# B&R Automation Studio project NAELD004C00R10L518F00 (part 25)

#### Local.var
```iecst
(*2023-02-13*)
(**)
(*Local Action, State & Status*)
VAR
	eAct : eMagRcpAction := MagRcpActIdle;
	eStat : eMagRcpAction := MagRcpActIdle;
	eStatus : eFBStatus := Idle;
	udiStatus : UDINT := 0;
	sStatTxt : STRING[200] := '';
	a_sStatText : ARRAY[0..50] OF STRING[200] := ['Idling','Creating Directory','Adding and Editing Files','Deleting Files','Get Info','Get List','Filtering Files','Reading Current Recipe','Loading Current Recipe','Writing Current Recipe Parameter','Saving List',40('')];
END_VAR
(**)
(*Local Alarm*)
VAR
	tyAlmData : tyAlmDat;
	a_tyAlmText : ARRAY[10000..10099] OF tyAlmTxt := [(sAlmText:='Create User Directory Error',sRcyText:='Unable To Create User Directory. Please Contact Nutek For A Possible Solution'),(sAlmText:='Create Magazine Recipe Directory Error',sRcyText:='Unable To Create Magazine Recipe Directory. Please Contact Nutek For A Possible Solution'),(sAlmText:='File Open Error While Adding & Editing',sRcyText:='An Error Was Encountered While Trying To Open File. Please Contact Nutek For A Possible Solution.'),(sAlmText:='File Create Error While Adding & Editing',sRcyText:='An Error Was Encountered While Trying To Create File. Please Contact Nutek For A Possible Solution.'),(sAlmText:='File Write Error While Adding & Editing',sRcyText:='An Error Was Encountered While Trying To Write File. Please Contact Nutek For A Possible Solution.'),(sAlmText:='File Close Error While Adding & Editing',sRcyText:='An Error Was Encountered While Trying To Close File. Please Contact Nutek For A Possible Solution.'),(sAlmText:='File Open Error While Deleting',sRcyText:='An Error Was Encountered While Trying To Open File. Please Contact Nutek For A Possible Solution.'),(sAlmText:='File Create Error While Deleting',sRcyText:='An Error Was Encountered While Trying To Create File. Please Contact Nutek For A Possible Solution.'),(sAlmText:='File Write Error While Deleting',sRcyText:='An Error Was Encountered While Trying To Write File. Please Contact Nutek For A Possible Solution.'),(sAlmText:='File Close Error While Deleting',sRcyText:='An Error Was Encountered While Trying To Close File. Please Contact Nutek For A Possible Solution.'),(sAlmText:='File Open Error While Getting List',sRcyText:='An Error Was Encountered While Trying To Open File. Please Contact Nutek For A Possible Solution.'),(sAlmText:='File Read Error While Getting List',sRcyText:='An Error Was Encountered While Trying To Read File. Please Contact Nutek For A Possible Solution.'),(sAlmText:='File Close Error While Getting List',sRcyText:='An Error Was Encountered While Trying To Close File. Please Contact Nutek For A Possible Solution.'),(sAlmText:='Directory Does Not Exist While Adding & Editing',sRcyText:='The Directory Does Not Exist.Please Contact Nutek For A Possible Solution.'),(sAlmText:='Directory Does Not Exist While Deleting',sRcyText:='The Directory Does Not Exist.Please Contact Nutek For A Possible Solution.'),(sAlmText:='File Open Error While Loading Current Recipe',sRcyText:='An Error Was Encountered While Trying To Open File. Please Contact Nutek For A Possible Solution.'),(sAlmText:='File Create Error While Loading Current Recipe',sRcyText:='An Error Was Encountered While Trying To Create File. Please Contact Nutek For A Possible Solution.'),(sAlmText:='File Write Error While Loading Current Recipe',sRcyText:='An Error Was Encountered While Trying To Write File. Please Contact Nutek For A Possible Solution.'),(sAlmText:='File Close Error While Loading Current Recipe',sRcyText:='An Error Was Encountered While Trying To Close File. Please Contact Nutek For A Possible Solution.'),(sAlmText:='Directory Does Not Exist While Loading Current Recipe',sRcyText:='The Directory Does Not Exist.Please Contact Nutek For A Possible Solution.'),(sAlmText:='File Open Error While Reading Current Recipe',sRcyText:='An Error Was Encountered While Trying To Open File. Please Contact Nutek For A Possible Solution.'),(sAlmText:='File Read Error While Reading Current Recipe',sRcyText:='An Error Was Encountered While Trying To Read File. Please Contact Nutek For A Possible Solution.'),(sAlmText:='File Close Error While Reading Current Recipe',sRcyText:='An Error Was Encountered While Trying To Close File. Please Contact Nutek For A Possible Solution.'),(sAlmText:='File Open Error While Writing Current Recipe Parameter',sRcyText:='An Error Was Encountered While Trying To Open File. Please Contact Nutek For A Possible Solution.'),(sAlmText:='File Create Error While Writing Current Recipe Parameter',sRcyText:='An Error Was Encountered While Trying To Create File. Please Contact Nutek For A Possible Solution.'),(sAlmText:='File Write Error While Writing Current Recipe Parameter',sRcyText:='An Error Was Encountered While Trying To Write File. Please Contact Nutek For A Possible Solution.'),(sAlmText:='File Close Error While Writing Current Recipe Parameter',sRcyText:='An Error Was Encountered While Trying To Close File. Please Contact Nutek For A Possible Solution.'),(sAlmText:='Directory Does Not Exist While Writing Current Recipe Parameter',sRcyText:='The Directory Does Not Exist.Please Contact Nutek For A Possible Solution.'),(sAlmText:='File Open Error While Saving List',sRcyText:='An Error Was Encountered While Trying To Open File. Please Contact Nutek For A Possible Solution.'),(sAlmText:='File Create Error While Saving List',sRcyText:='An Error Was Encountered While Trying To Create File. Please Contact Nutek For A Possible Solution.'),(sAlmText:='File Write Error While Saving List',sRcyText:='An Error Was Encountered While Trying To Write File. Please Contact Nutek For A Possible Solution.'),(sAlmText:='File Close Error While Saving List',sRcyText:='An Error Was Encountered While Trying To Close File. Please Contact Nutek For A Possible Solution.'),(sAlmText:='Directory Does Not Exist While Saving List',sRcyText:='The Directory Does Not Exist.Please Contact Nutek For A Possible Solution.'),67(0)];
END_VAR
(**)
(*Local Output*)
VAR
	bNmExist : BOOL;
	bNmNotExist : BOOL;
	bNmEmpty : BOOL;
	bListFull : BOOL;
	a_tyCurrList : ARRAY[1..c_udiMagRcpMax] OF tyMagRcpParam;
	a_tyFilterList : ARRAY[1..c_udiMagRcpMax] OF tyMagRcpParam;
	a_tySortList : ARRAY[1..c_udiMagRcpMax] OF tyMagRcpParam;
	tyTempList : tyMagRcpParam;
	tyInfoOut : tyMagRcpParam;
	bFileNotFound : BOOL;
	tyCurrRcp : tyMagRcpParam;
END_VAR
(**)
(*Local Input*)
VAR
	udiRstErr : UDINT := 0;
	bPrep : BOOL := FALSE;
	bDis : BOOL := FALSE;
	dtCurrDT : DATE_AND_TIME;
	sSearch : STRING[254] := '';
	tyInfoIn : tyMagRcpParam;
	tyCurrRcpWr : tyMagRcpParam;
	sListFileName : STRING[80] := 'MagazineRecipeList.dat';
	sSingleFileName : STRING[80] := 'MagazineRecipe.dat';
	sProgNm : STRING[15] := 'MagRcp';
	bNtSettingsLoadDone : BOOL := TRUE;
	udiSortCurrenTotalCntr : UDINT;
	iSortCurrentInnerCntr : INT;
	iSortCurrentOuterCntr : INT;
	iTotalRcp : INT;
	i : {REDUND_UNREPLICABLE} INT;
	udi : UDINT;
	sDebug : STRING[300];
	tyTempRecipe : tyMagRcpParam;
END_VAR
(**)
(*Local*)
VAR
	bRstErr : BOOL;
	udiRstErrOld : UDINT;
	bInitDone : BOOL;
	bInitialDone : BOOL;
	usiStep : USINT;
	udiAddStatus : UDINT;
	a_tyListTemp : ARRAY[1..c_udiMagRcpMax] OF tyMagRcpParam;
	fbDirCreate1 : fbDirCreate;
	fbDirCreate2 : fbDirCreate;
	fbFileReadList : fbFileFullRead;
	fbFileWriteList : fbFileFullWrite;
	fbFileReadSingle : fbFileFullRead;
	fbFileWriteSingle : fbFileFullWrite;
	fbFileLoadSingle : fbFileFullWrite;
	iFilterCtr : INT;
	udiModuleNum : UDINT := 4901;
END_VAR
```

#### Act_Alarm.st
```iecst
(** 2019-03-25 **)
ACTION Act_Alarm:

	//Error
	IF EDGEPOS(eStatus = Error) THEN

		tyAlmData.sProgNm		:= p_sProgNm;
		tyAlmData.udiCode		:= udiStatus;
		tyAlmData.eSeverity		:= AlmSeverityError;
		tyAlmData.udiRunTime	:= tyAlmData.udiRunTime + 1;
		tyAlmData.bAlm			:= TRUE;
		tyAlmData.udiModuleNum  := udiModuleNum;
		g_sMagRcpProgNm			:= p_sProgNm;
		//Get Error Message
		IF tyAlmData.udiCode < 10000 OR tyAlmData.udiCode > 10099 THEN
			tyAlmData.sAlmMsg	:= 'Unknown';
			tyAlmData.sRcyMsg	:= 'Unknown';
		ELSE
			tyAlmData.sAlmMsg	:= a_tyAlmText[tyAlmData.udiCode].sAlmText;
			tyAlmData.sRcyMsg	:= a_tyAlmText[tyAlmData.udiCode].sRcyText;
		END_IF

		sStatTxt	:= tyAlmData.sAlmMsg;

	ELSIF bRstErr AND (tyAlmData.udiCode <> 0) THEN

		tyAlmData.udiCode	:= 0;
		tyAlmData.eSeverity	:= AlmSeverityNA;
		tyAlmData.sAlmMsg	:= '';
		tyAlmData.sRcyMsg	:= '';
		tyAlmData.bAlm			:= FALSE;
		sStatTxt	:= a_sStatText[eStat];

	END_IF

END_ACTION
```

#### Act_InitGlobal.st
```iecst
(** 2019-03-25 **)
ACTION Act_InitGlobal:

	(* Always Change If Project Change *)

	//Pass Data To Link
	p_bLinkStartupRun ACCESS p_StartupRun;

	//Pass Data To Internal Use
	p_udiRstErr ACCESS p_RstErrReset;
	p_dtCurrDT ACCESS p_TimeCurrDT;
	p_sSearch ACCESS p_UIMagRcpSearch1;
	p_tyInfoIn ACCESS p_UIMagRcpInfoIn1;
	p_sListFileName ACCESS p_NtParamMagRcpListFileNm1;
	p_sSingleFileName ACCESS p_NtParamMagRcpSingleFileNm1;
	p_sProgNm ACCESS p_NtParamMagRcpProgNm1;
	p_bNtSettingsLoadDone ACCESS p_StartupNtSettingsLoadDone;

	(* Always Change If Project Change *)

END_ACTION
```

#### Act_Initial.st
```iecst
(** 2019-05-07 **)
ACTION Act_Initial:

	//Initial
	sStatTxt	:= a_sStatText[eStat];

	fbDirCreate1.sDevice	:= 'F';
	fbDirCreate1.sDirName	:= 'User';
	fbDirCreate1(bEn := FALSE);

	fbDirCreate2.sDevice	:= 'User';
	fbDirCreate2.sDirName	:= 'MagazineRecipe1';
	fbDirCreate2(bEn := FALSE);

	fbFileReadList.sDevice			:= 'MagRcp1';
	fbFileReadList.sFile			:= p_sListFileName;
	fbFileReadList.udiOffset		:= 0;
	fbFileReadList.p_Dest			:= ADR(a_tyCurrList);
	fbFileReadList.udiLen			:= SIZEOF(a_tyCurrList);
	fbFileReadList(bEn := FALSE);

	fbFileWriteList.sDevice			:= 'MagRcp1';
	fbFileWriteList.sFile			:= p_sListFileName;
	fbFileWriteList.udiOffset		:= 0;
	fbFileWriteList.p_Src			:= ADR(a_tyListTemp);
	fbFileWriteList.udiLen			:= SIZEOF(a_tyListTemp);
	fbFileWriteList.udiOption		:= 0;
	fbFileWriteList(bEn := FALSE);

	fbFileReadSingle.sDevice		:= 'MagRcp1';
	fbFileReadSingle.sFile			:= p_sSingleFileName;
	fbFileReadSingle.udiOffset		:= 0;
	fbFileReadSingle.p_Dest			:= ADR(tyCurrRcp);
	fbFileReadSingle.udiLen			:= SIZEOF(tyCurrRcp);
	fbFileReadSingle(bEn := FALSE);

	fbFileLoadSingle.sDevice		:= 'MagRcp1';
	fbFileLoadSingle.sFile			:= p_sSingleFileName;
	fbFileLoadSingle.udiOffset		:= 0;
	fbFileLoadSingle.p_Src			:= ADR(tyCurrRcp);
	fbFileLoadSingle.udiLen			:= SIZEOF(tyCurrRcp);
	fbFileLoadSingle.udiOption		:= 0;
	fbFileLoadSingle(bEn := FALSE);

	fbFileWriteSingle.sDevice		:= 'MagRcp1';
	fbFileWriteSingle.sFile			:= p_sSingleFileName;
	fbFileWriteSingle.udiOffset		:= 0;
	fbFileWriteSingle.p_Src			:= ADR(p_tyCurrRcpWr);
	fbFileWriteSingle.udiLen		:= SIZEOF(p_tyCurrRcpWr);
	fbFileWriteSingle.udiOption		:= 0;
	fbFileWriteSingle(bEn := FALSE);

END_ACTION
```

#### Act_LinkAction.st
```iecst
(** 2019-03-29 **)
ACTION Act_LinkAction:

	IF p_bLinkStartupRun = TRUE THEN
		p_eAct ACCESS p_StartupMagRcpAct1;
	ELSE
		p_eAct ACCESS p_UIMagRcpAct1;
	END_IF

END_ACTION
```

#### Init.st
```iecst
(** 2019-05-04 **)
PROGRAM _INIT

	(* Always Change If Project Change *)

	//Pass Address To Global Address For External Use
	//Action, State & Status
	p_MagRcpStat1	:= ADR(eStat);
	p_MagRcpStatus1	:= ADR(eStatus);
	p_MagRcpStatTxt1	:= ADR(sStatTxt);

	//Alarm
	p_MagRcpAlmData1	:= ADR(tyAlmData);

	//Output
	p_MagRcpNmExist1		:= ADR(bNmExist);
	p_MagRcpNmNotExist1		:= ADR(bNmNotExist);
	p_MagRcpNmEmpty1		:= ADR(bNmEmpty);
	p_MagRcpListFull1		:= ADR(bListFull);
	p_MagRcpCurrList1		:= ADR(a_tyCurrList);
	p_MagRcpFilterList1		:= ADR(a_tyFilterList);
	p_MagRcpSortedList1		:= ADR(a_tySortList);
	p_MagRcpInfoOut1		:= ADR(tyInfoOut);
	p_MagRcpFileNotFound1	:= ADR(bFileNotFound);

	p_MagRcpCurrRcp1				:= ADR(tyCurrRcp);
	p_MagRcpCurrRcpNm1				:= ADR(tyCurrRcp.sRcpNm);
	p_MagRcpCurrRcpTtlSlt1			:= ADR(tyCurrRcp.diTtlSlt);
	p_MagRcpCurrRcpSltToSlt1		:= ADR(tyCurrRcp.diSltToSltInUM);
	p_MagRcpCurrRcpMag1Slt1Pos1		:= ADR(tyCurrRcp.diMag1Slt1PosInUM);
	p_MagRcpCurrRcpMag2Slt1Pos1		:= ADR(tyCurrRcp.diMag2Slt1PosInUM);
	p_MagRcpCurrRcpMag3Slt1Pos1		:= ADR(tyCurrRcp.diMag3Slt1PosInUM);
	p_MagRcpCurrRcpMag4Slt1Pos1		:= ADR(tyCurrRcp.diMag4Slt1PosInUM);
	p_MagRcpCurrRcpMag1TravPos1		:= ADR(tyCurrRcp.diMag1TravPosInUM);
	p_MagRcpCurrRcpMag2TravPos1		:= ADR(tyCurrRcp.diMag2TravPosInUM);
	p_MagRcpCurrRcpMag3TravPos1		:= ADR(tyCurrRcp.diMag3TravPosInUM);
	p_MagRcpCurrRcpMag4TravPos1		:= ADR(tyCurrRcp.diMag4TravPosInUM);
	p_MagRcpCurrRcpDisplayInfo1		:= ADR(tyCurrRcp.sDisplayInfo);
	p_MagRcpCurrRcpLastModified1	:= ADR(tyCurrRcp.dtLastModified);
	p_MagRcpCurrRcpMagMaxBrdWidth1	:= ADR(tyCurrRcp.diMagMaxBrdWidth);
	p_MagRcpCurrRcpMagModel1		:= ADR(tyCurrRcp.usiMagModel);
	p_MagRcpCurrRcpSBarDisabled1	:= ADR(tyCurrRcp.bSafetyBarDisabled);
	p_MagRcpCurrRcpMagHeightChkEn1	:= ADR(tyCurrRcp.bMagHeightChkEn);
	(* Always Change If Project Change *)

END_PROGRAM
```

### McParam.typ
```iecst
(*2019-05-04*)
(**)
(*Action*)

TYPE
	eMcParamAction :
		(
		McParamActIdle,
		McParamActCreateDir,
		McParamActRead,
		McParamActWrite
		);
END_TYPE

(**)
(*Data*)

TYPE
	tyMcParam : 	STRUCT
		a_bLFOnline : ARRAY[1..c_diLFClntNum]OF BOOL;
		a_sLFIPAddr : ARRAY[1..c_diLFClntNum]OF STRING[15];
		sMcNm : STRING[30] := 'Triple Magazine Line Loader';
		uiSSaverTmInSec : UINT := 1800;
		bSSaverEn : BOOL := FALSE;
		usiDefaultMcMod : USINT := 0;
		usiDefaultFlippedBrd : USINT := 0;
		diAWPusherAtHmPosInUM : DINT;
		bAWPusherDis : BOOL := FALSE;
		diWidthAtHmPosInUM : DINT;
		diConvInitTmInMS : DINT := 6000;
		diTranOutErrDlyTmInMS : DINT := 12000;
		diMag1ConvRunTmOutInMS : DINT := 20000;
		diMag2ConvRunTmOutInMS : DINT := 20000;
		diMag3ConvRunTmOutInMS : DINT := 20000;
		diMag4ConvRunTmOutInMS : DINT := 20000;
		diTravPosA : DINT;
		diTravPosB : DINT;
		diLifterPosA : DINT;
		diLifterPosB : DINT;
		bAWDis : BOOL := FALSE;
		bMnlAccDat : BOOL := FALSE;
		bAutoStepEn : BOOL := FALSE;
		bVSMEMAEn : BOOL := TRUE;
		bChgParamEn : BOOL := TRUE;
		bHermesRmtEn : BOOL := FALSE;
		bLongBrdEn : BOOL := FALSE;
		bOutShutterDis : BOOL := FALSE;
		bLFEn : BOOL := FALSE;
		bLCSLFEn : BOOL := FALSE;
		bLCSReqRcpEn : BOOL := FALSE;
		bLCSManageRcpEn : BOOL := FALSE;
		bLCSLiveDatEn : BOOL := FALSE;
		bLFLeaderMc : BOOL := FALSE;
		bSectionLeader : BOOL := FALSE;
		bDSWidthChkEn : BOOL := FALSE;
		diLFMcIdxBeforeOven : DINT := 1;
		diLFMcIdxAfterOven : DINT := 1;
		diLFMcIdxBeforeOven2 : DINT := 1;
		diLFMcIdxAfterOven2 : DINT := 1;
		usiLang : USINT := 0;
		tyLftSenAntiGapDly : tyAntiGapDly := (diSigOnTm:=0,diSigOffTm:=0);
		tyRgtSenAntiGapDly : tyAntiGapDly := (diSigOnTm:=0,diSigOffTm:=500);
		tyMagConvEntrySenAntiGapDly : tyAntiGapDly := (diSigOnTm:=100,diSigOffTm:=100);
		tyMagConvPresentSenAntiGapDly : tyAntiGapDly := (diSigOnTm:=1000,diSigOffTm:=100);
		eDSCommA : eMcSetCommMod := McSetCommModSMEMA;
		tyDSCommASMEMA : tySMEMAParam := (eSelection:=SMEMASelIPC9851,bStatSigSetGd:=FALSE);
		eDSCommB : eMcSetCommMod := McSetCommModSMEMA;
		tyDSCommBSMEMA : tySMEMAParam := (eSelection:=SMEMASelIPC9851,bStatSigSetGd:=FALSE);
		diWidthOffsetInUM : DINT := 0;
		diMagAutoDetectSenTmInMS : DINT := 2000;
		bAGVComEn : BOOL := FALSE;
		bAutoLogoutEn : BOOL := FALSE;
		diAutoLogoutTmInSec : DINT := 60000;
		sIPAddr : STRING[15] := '192.168.0.32';
		sSubnetMask : STRING[15] := '255.255.255.0';
		eNetworkMod : eNetworkConfigMod := SetIPManually;
		bLFSeqStayActive : BOOL := FALSE;
		bLFBuzMute : BOOL := FALSE;
		bScannerEn : BOOL := TRUE;
		diVID : DINT := 1529;
		diPID : DINT := 8716;
		eAGVComProtocol : eMcAGVCommProtocol := McSetAGVCommOPCUA;
		eMagExMode : eMcMagExchangeMode := McSetMagXcAutoManMode;
		bAIVSizeDisabled : BOOL := FALSE;
		diRS232StartCode1 : DINT := -1;
		diRS232StartCode2 : DINT := -1;
		diRS232EndCode1 : DINT := -1;
		diRS232EndCode2 : DINT := -1;
		diTravOutletFixtoFixPos : DINT := 0;
		bDisableFMWarning : BOOL := FALSE;
		bDBAOnWOAlign : BOOL := FALSE;
		diLMCfbTmInMS : DINT := 20000;
		bMagWidthChkDis : BOOL := FALSE;
		diMag1WidthChkDetDist : DINT := 3000;
		diMag2WidthChkDetDist : DINT := 3000;
		diMag3WidthChkDetDist : DINT := 3000;
		bDBAOnRgtSen : BOOL := FALSE;
		bHermesSvyEn : BOOL := FALSE;
		bHermesScannerEn : BOOL := TRUE;
		bMesRFIDEn : BOOL := FALSE;
		diMesRFIDTOInMS : DINT := 5000;
		diTravLaneBOffset : DINT := 0;
	END_STRUCT;
END_TYPE

(**)

TYPE
	tyAntiGapDly : 	STRUCT
		diSigOnTm : DINT;
		diSigOffTm : DINT;
	END_STRUCT;
	eMcSetCommMod :
		(
		McSetCommModSMEMA,
		McSetCommModHermes
		);
	eMcAGVCommProtocol :
		(
		McSetAGVCommOPCUA,
		McSetAGVCommHardIO,
		McSetAGVCommDisabled
		);
	eMcMagExchangeMode :
		(
		McSetMagXcAutoManMode,
		McSetMagXcAutoMode,
		McSetMagXcManMode
		);
END_TYPE
```

### McParam.var
```iecst
(*2019-04-17*)
(**)
(*Action & State & Status*)
VAR
	p_McParamStat : UDINT;
	p_McParamStatus : UDINT;
	p_McParamStatTxt : UDINT;
END_VAR
(**)
(*Alarm*)
VAR
	p_McParamAlmData : UDINT;
END_VAR
(**)
(*Output*)
VAR
	p_McParamFileNotFound : UDINT;
END_VAR
(**)
VAR
	p_McParamCurr : UDINT;
END_VAR
(**)
VAR
	p_McParamLFOnline : UDINT;
	p_McParamLFIPAddr : UDINT;
END_VAR
(**)
VAR
	p_McParamMcNm : UDINT;
	p_McParamSSaverTm : UDINT;
	p_McParamSSaverEn : UDINT;
	p_McParamDefaultMcMod : UDINT;
	p_McParamDefaultFlippedBrd : UDINT;
	p_McParamWidthAtHmPos : UDINT;
	p_McParamConvInitTm : UDINT;
	p_McParamTranOutErrDlyTm : UDINT;
	p_McParamMag1ConvRunTmOut : UDINT;
	p_McParamMag2ConvRunTmOut : UDINT;
	p_McParamMag3ConvRunTmOut : UDINT;
	p_McParamMag4ConvRunTmOut : UDINT;
	p_McParamTravPosA : UDINT;
	p_McParamTravPosB : UDINT;
	p_McParamLifterPosA : UDINT;
	p_McParamLifterPosB : UDINT;
	p_McParamAWDis : UDINT;
	p_McParamMnlAccDat : UDINT;
	p_McParamAutoStepEn : UDINT;
	p_McParamVSMEMAEn : UDINT;
	p_McParamChgParamEn : UDINT;
	p_McParamHermesRmtEn : UDINT;
	p_McParamLongBrdEn : UDINT;
	p_McParamOutShutterDis : UDINT;
	p_McParamMagAutoDetTm : UDINT;
	p_McParamAGVComEn : UDINT;
END_VAR
(**)
VAR
	p_McParamLFEn : UDINT;
	p_McParamLCSLFEn : UDINT;
	p_McParamLCSReqRcpEn : UDINT;
	p_McParamLCSManageRcpEn : UDINT;
	p_McParamLCSLiveDatEn : UDINT;
	p_McParamLFLeaderMc : UDINT;
	p_McParamSectionLeader : UDINT;
	p_McParamDSWidthChkEn : UDINT;
	p_McParamLFMcIdxBeforeOven : UDINT;
	p_McParamLFMcIdxAfterOven : UDINT;
	p_McParamLFMcIdxBeforeOven2 : UDINT;
	p_McParamLFMcIdxAfterOven2 : UDINT;
END_VAR
(**)
VAR
	p_McParamLang : UDINT;
END_VAR
(**)
VAR
	p_McParamConvLftSenAntiGap : UDINT;
	p_McParamConvLftSenOnTm : UDINT;
	p_McParamConvLftSenOffTm : UDINT;
	p_McParamConvRgtSenAntiGap : UDINT;
	p_McParamConvRgtSenOnTm : UDINT;
	p_McParamConvRgtSenOffTm : UDINT;
	p_McParamMagConvEntrySenAntiGap : UDINT;
	p_McParamMagConvEntrySenOnTm : UDINT;
	p_McParamMagConvEntrySenOffTm : UDINT;
	p_McParamMagConvPresentAntiGap : UDINT;
	p_McParamMagConvPresentSenOnTm : UDINT;
	p_McParamMagConvPresentSenOffTm : UDINT;
END_VAR
(**)
VAR
	p_McParamDSCommAMod : UDINT;
	p_McParamDSSMEMAAParam : UDINT;
	p_McParamDSSMEMAASelection : UDINT;
	p_McParamDBAAStatSetGd : UDINT;
END_VAR
(**)
VAR
	p_McParamDSCommBMod : UDINT;
	p_McParamDSSMEMABParam : UDINT;
	p_McParamDSSMEMABSelection : UDINT;
	p_McParamDBABStatSetGd : UDINT;
END_VAR
(**)
VAR
	p_McParamAIVComm : UDINT;
	p_McParamAIVSvrPort : UDINT;
	p_McParamAIVClientPort : UDINT;
	p_McParamAIVClientAddr : UDINT;
END_VAR
(**)
VAR
	p_McParamWidthOffset : UDINT;
	p_McParamNetworkMod : UDINT;
END_VAR
(**)
VAR
	p_McParamLFSeqStayActive : UDINT;
	p_McParamLFBuzMute : UDINT;
END_VAR
(*USB Barcode Reader*)
VAR
	p_McParamVID : UDINT;
	p_McParamPID : UDINT;
	p_McParamScannerEn : UDINT;
	p_McParamAGVComProtocol : UDINT;
	p_McParamMagExMode : UDINT;
END_VAR
(**)
VAR
	p_McParamRS232StartCode1 : UDINT;
	p_McParamRS232StartCode2 : UDINT;
	p_McParamRS232EndCode1 : UDINT;
	p_McParamRS232EndCode2 : UDINT;
END_VAR
(**)
VAR
	p_McParamAWPusherAtHmPos : UDINT;
	p_McParamAWPusherDis : UDINT;
END_VAR
(**)
(**)
VAR
	p_McParamTravOutletFixtoFixPos : UDINT;
	p_McParamDisableFMWarning : UDINT;
END_VAR
(**)
VAR
	p_McParamDBAOnWOAlign : UDINT;
	p_McParamMagWidthChkDis : UDINT;
	p_McParamMag1WidthChkDetDist : UDINT;
	p_McParamMag2WidthChkDetDist : UDINT;
	p_McParamMag3WidthChkDetDist : UDINT;
	p_McParamDBAOnRgtSen : UDINT;
END_VAR
(**)
VAR
	p_McParamHermesSvyEn : UDINT;
	p_McParamHermesScannerEn : UDINT;
	p_McParamMesRFIDEn : UDINT;
	p_McParamMesRFIDTOInMS : UDINT;
	p_McParamTravLaneBOffset : UDINT;
END_VAR
```

### Program Logical/McParam/McParam

#### InputRef.var
```iecst
(*2019-03-25*)
(**)
(*General*)
VAR
	p_eAct : REFERENCE TO eMcParamAction;
	p_udiRstErr : REFERENCE TO UDINT;
END_VAR
(**)
(*Configuration*)
VAR
	p_sFileName : REFERENCE TO STRING[80];
	p_tyMcParamWr : REFERENCE TO tyMcParam;
	p_sProgNm : REFERENCE TO STRING[15];
	p_bNtSettingsLoadDone : REFERENCE TO BOOL;
	p_bRmtHermesWriteConfig : REFERENCE TO BOOL;
	p_bSvyHermesWriteConfig : REFERENCE TO BOOL;
	p_tyHermesConfigurationWr : REFERENCE TO tyHermesConfiguration;
	p_bNtParamProjLaneBPrep : REFERENCE TO BOOL;
	p_eNtParamCustomerReq : REFERENCE TO eCustomer;
END_VAR
```

#### Local.var
```iecst
(*2019-04-30*)
(**)
(*Local Action, State & Status*)
VAR
	eAct : eMcParamAction := McParamActIdle;
	eStat : eMcParamAction := McParamActIdle;
	eStatus : eFBStatus := Idle;
	udiStatus : UDINT := 0;
	sStatTxt : STRING[200] := '';
	a_sStatText : ARRAY[0..50] OF STRING[200] := ['Idling','Creating Directory','Reading Files','Writing Files',47('')];
END_VAR
(**)
(*Local Alarm*)
VAR
	tyAlmData : tyAlmDat;
	a_tyAlmText : ARRAY[10000..10099] OF tyAlmTxt := [(sAlmText:='Create User Directory Error',sRcyText:='Unable To Create User Directory. Please Contact Nutek For A Possible Solution'),(sAlmText:='Create Machine Parameter Directory Error',sRcyText:='Unable To Create Machine Parameter Directory. Please Contact Nutek For A Possible Solution'),(sAlmText:='File Open Error While Writing',sRcyText:='An Error Was Encountered While Trying To Open File. Please Contact Nutek For A Possible Solution.'),(sAlmText:='File Create Error While Writing',sRcyText:='An Error Was Encountered While Trying To Create File. Please Contact Nutek For A Possible Solution.'),(sAlmText:='File Write Error',sRcyText:='An Error Was Encountered While Trying To Write File. Please Contact Nutek For A Possible Solution.'),(sAlmText:='File Close Error While Writing',sRcyText:='An Error Was Encountered While Trying To Close File. Please Contact Nutek For A Possible Solution.'),(sAlmText:='File Open Error While Reading',sRcyText:='An Error Was Encountered While Trying To Open File. Please Contact Nutek For A Possible Solution.'),(sAlmText:='File Read Error',sRcyText:='An Error Was Encountered While Trying To Read File. Please Contact Nutek For A Possible Solution.'),(sAlmText:='File Close Error While Reading',sRcyText:='An Error Was Encountered While Trying To Close File. Please Contact Nutek For A Possible Solution.'),(sAlmText:='Directory Does Not Exist While Writing',sRcyText:='The Directory Does Not Exist.Please Contact Nutek For A Possibe Solution.'),90(0)];
END_VAR
(**)
(*Local Output*)
VAR
	tyMcParamCurr : tyMcParam;
	bFileNotFound : BOOL;
END_VAR
(**)
(*Local Input*)
VAR
	udiRstErr : UDINT := 0;
	sFileName : STRING[80] := 'MachineParameter.dat';
	tyMcParamWr : tyMcParam;
	sProgNm : STRING[15] := 'McParam';
	bNtSettingsLoadDone : BOOL := TRUE;
END_VAR
(**)
(*Local*)
VAR
	bRstErr : BOOL;
	udiRstErrOld : UDINT;
	bInitDone : BOOL;
	bInitialDone : BOOL;
	usiStep : USINT;
	tyMcParamTemp : tyMcParam;
	fbDirCreate1 : fbDirCreate;
	fbDirCreate2 : fbDirCreate;
	fbFileRead1 : fbFileFullRead;
	fbFileWrite1 : fbFileFullWrite;
	fbFileWrite2 : fbFileFullWrite;
	udiModuleNum : UINT := 5251;
END_VAR
(*//ADD*)
VAR
	sHMIIPAddr : STRING[15];
	sVNCIPAddr : STRING[15];
	uiNSIdx : UINT;
	fbConnectOPCUA : fbOPCUAConnect;
	fbDisconnectOPCUA : fbOPCUADisconnect;
	dwConnectionHdl : DWORD;
	sHMIAddrNodeID : STRING[15];
	sVNCAddrNodeID : STRING[5];
	fbReadGetNodeHdlList : fbOPCUAGetNodeHdlList;
	fbReadList : fbOPCUAReadList;
	tyReadHdls : tyOPCUAHdlList;
	fbWriteGetNodeHdlList : fbOPCUAGetNodeHdlList;
	fbWriteList : fbOPCUAWriteList;
	tyWriteHdls : tyOPCUAHdlList;
	sObjIDNodeID : STRING[5];
	sSaveCfgNodeID : STRING[5];
	fbSaveCfgMethodGetHdl : fbOPCUAMethodGetHandle;
	fbSaveCfgMethodCall : fbOPCUAMethodCall;
	sLoadCfgNodeID : STRING[5];
	fbLoadCfgMethodGetHdl : fbOPCUAMethodGetHandle;
	fbLoadCfgMethodCall : fbOPCUAMethodCall;
	dwMethodHdl : DWORD;
	usiChkIpAddrStep : USINT;
	bWarning : BOOL;
	bConnected : BOOL;
END_VAR
```

#### Act_Alarm.st
```iecst
(** 2019-03-25 **)
ACTION Act_Alarm:

	//Error
	IF EDGEPOS(eStatus = Error) THEN

		tyAlmData.sProgNm		:= p_sProgNm;
		tyAlmData.udiCode		:= udiStatus;
		tyAlmData.eSeverity		:= AlmSeverityError;
		tyAlmData.udiRunTime	:= tyAlmData.udiRunTime + 1;
		tyAlmData.bAlm			:= TRUE;
		tyAlmData.udiModuleNum  := udiModuleNum;
		g_sMcParamProgNm		:= p_sProgNm;

		//Get Error Message
		IF tyAlmData.udiCode < 10000 OR tyAlmData.udiCode > 10099 THEN
			tyAlmData.sAlmMsg	:= 'Unknown';
			tyAlmData.sRcyMsg	:= 'Unknown';
		ELSE
			tyAlmData.sAlmMsg	:= a_tyAlmText[tyAlmData.udiCode].sAlmText;
			tyAlmData.sRcyMsg	:= a_tyAlmText[tyAlmData.udiCode].sRcyText;
		END_IF

		sStatTxt	:= tyAlmData.sAlmMsg;
	ELSIF bConnected = FALSE THEN
		tyAlmData.sProgNm		:= p_sProgNm;
		tyAlmData.udiCode		:= udiStatus;
		tyAlmData.eSeverity		:= AlmSeverityWarning;
		tyAlmData.udiRunTime	:= tyAlmData.udiRunTime + 1;
		tyAlmData.bWarning			:= TRUE;
		tyAlmData.udiModuleNum  := udiModuleNum;
		g_sMcParamProgNm		:= p_sProgNm;

		//Get Error Message
		IF tyAlmData.udiCode < 10000 OR tyAlmData.udiCode > 10099 THEN
			tyAlmData.sAlmMsg	:= 'Unknown';
			tyAlmData.sRcyMsg	:= 'Unknown';
		ELSE
			tyAlmData.sAlmMsg	:= a_tyAlmText[tyAlmData.udiCode].sAlmText;
			tyAlmData.sRcyMsg	:= a_tyAlmText[tyAlmData.udiCode].sRcyText;
		END_IF

		sStatTxt	:= tyAlmData.sAlmMsg;
	ELSIF bRstErr AND (tyAlmData.udiCode <> 0) THEN

		tyAlmData.udiCode	:= 0;
		tyAlmData.eSeverity	:= AlmSeverityNA;
		tyAlmData.sAlmMsg	:= '';
		tyAlmData.sRcyMsg	:= '';
		tyAlmData.bAlm			:= FALSE;
		tyAlmData.bWarning			:= FALSE;
		sStatTxt	:= a_sStatText[eStat];

	END_IF

END_ACTION
```

#### Act_InitGlobal.st
```iecst
(** 2019-03-25 **)
ACTION Act_InitGlobal:

	(* Always Change If Project Change *)

	//Pass Data To Link
	p_bLinkStartupRun ACCESS p_StartupRun;

	//Pass Data To Internal Use
	p_udiRstErr ACCESS p_RstErrReset;
	p_sFileName ACCESS p_NtParamMcParamFileNm;
	p_tyMcParamWr ACCESS p_UIMcParamWr;
	p_sProgNm ACCESS p_NtParamMcParamProgNm;
	p_bNtSettingsLoadDone ACCESS p_StartupNtSettingsLoadDone;
	p_bRmtHermesWriteConfig ACCESS p_RmtHermesWriteConfig; //new for Hermes 1.3
	p_bSvyHermesWriteConfig ACCESS p_SvyHermesWriteConfig; //new for Hermes 1.3
	p_tyHermesConfigurationWr ACCESS p_HermesConfigurationWr; //new for Hermes 1.3
	p_bNtParamProjLaneBPrep ACCESS p_NtParamProjLaneBPrep;
	p_eNtParamCustomerReq ACCESS p_NtParamCustomerReq;
	(* Always Change If Project Change *)

END_ACTION
```

#### Act_Initial.st
```iecst
(** 2019-01-15 **)
ACTION Act_Initial:

	//Initial
	sStatTxt	:= a_sStatText[eStat];

	fbDirCreate1.sDevice	:= 'F';
	fbDirCreate1.sDirName	:= 'User';
	fbDirCreate1(bEn := FALSE);

	fbDirCreate2.sDevice	:= 'User';
	fbDirCreate2.sDirName	:= 'MachineParameter';
	fbDirCreate2(bEn := FALSE);

	fbFileRead1.sDevice			:= 'McParam';
	fbFileRead1.sFile			:= p_sFileName;
	fbFileRead1.udiOffset		:= 0;
	fbFileRead1.p_Dest			:= ADR(tyMcParamCurr);
	fbFileRead1.udiLen			:= SIZEOF(tyMcParamCurr);
	fbFileRead1(bEn := FALSE);

	fbFileWrite1.sDevice		:= 'McParam';
	fbFileWrite1.sFile			:= p_sFileName;
	fbFileWrite1.udiOffset		:= 0;
	fbFileWrite1.p_Src			:= ADR(p_tyMcParamWr);
	fbFileWrite1.udiLen			:= SIZEOF(p_tyMcParamWr);
	fbFileWrite1.udiOption		:= 0;
	fbFileWrite1(bEn := FALSE);

	fbFileWrite2.sDevice		:= 'McParam';
	fbFileWrite2.sFile			:= p_sFileName;
	fbFileWrite2.udiOffset		:= 0;
	fbFileWrite2.p_Src			:= ADR(tyMcParamTemp);
	fbFileWrite2.udiLen			:= SIZEOF(tyMcParamTemp);
	fbFileWrite2.udiOption		:= 0;
	fbFileWrite2(bEn := FALSE);

	//ADDED
	sVNCAddrNodeID := '54267'; // HMI VNC's IP Address Node ID
	sHMIAddrNodeID := '54248'; // HMI Network's IP Address Node ID
	sObjIDNodeID := '54159'; // HMI MethodSet's Node ID
	sSaveCfgNodeID := '54322'; // HMI Save Method's Node ID
	sLoadCfgNodeID := '54321'; // HMI Load Method's Node ID

	uiNSIdx := 4;
	fbConnectOPCUA.tyOPCUAParam.sPort := '4841';
	fbConnectOPCUA(bEn := FALSE);
	fbReadGetNodeHdlList.usiNSIdx := uiNSIdx;
	fbReadGetNodeHdlList.uiTagNmCnt := 2;
	fbReadGetNodeHdlList.a_sServerTagNm[0] := sVNCAddrNodeID;
	fbReadGetNodeHdlList.a_sServerTagNm[1] := sHMIAddrNodeID;
	fbReadGetNodeHdlList(bEn := FALSE);
	fbReadList.uiTagNmCnt := 2;
	fbReadList(bEn := FALSE);

	fbWriteGetNodeHdlList.usiNSIdx := uiNSIdx;
	fbWriteGetNodeHdlList.uiTagNmCnt := 2;
	fbWriteGetNodeHdlList.a_sServerTagNm[0] := sVNCAddrNodeID;
	fbWriteGetNodeHdlList.a_sServerTagNm[1] := sHMIAddrNodeID;
	fbWriteGetNodeHdlList(bEn := FALSE);
	fbWriteList.uiTagNmCnt := 2;
	fbWriteList(bEn := FALSE);

	fbSaveCfgMethodGetHdl.uiNSIdx := uiNSIdx;
	fbSaveCfgMethodGetHdl.sObjectIdentifier := sObjIDNodeID;
	fbSaveCfgMethodGetHdl.sMethodIdentifier := sSaveCfgNodeID;
	fbSaveCfgMethodGetHdl(bEn := FALSE);
	fbSaveCfgMethodCall(bEn := FALSE);

	fbLoadCfgMethodGetHdl.uiNSIdx := uiNSIdx;
	fbLoadCfgMethodGetHdl.sObjectIdentifier := sObjIDNodeID;
	fbLoadCfgMethodGetHdl.sMethodIdentifier := sLoadCfgNodeID;
	fbLoadCfgMethodGetHdl(bEn := FALSE);
	fbLoadCfgMethodCall(bEn := FALSE);

	fbDisconnectOPCUA(bEn := FALSE);
END_ACTION
```

#### Act_InitLocal.st
```iecst
(** 2019-03-25 **)
ACTION Act_InitLocal:

	//Input Reference Link To Local Variable
	p_eAct ACCESS ADR(eAct);
	p_udiRstErr ACCESS ADR(udiRstErr);
	p_sFileName ACCESS ADR(sFileName);
	p_tyMcParamWr ACCESS ADR(tyMcParamWr);
	p_sProgNm ACCESS ADR(sProgNm);
	p_bNtSettingsLoadDone ACCESS ADR(bNtSettingsLoadDone);

	//ADD
	p_bAlarmWarning ACCESS ADR(bWarning);
END_ACTION
```

#### Act_Link.st
```iecst
(** 2021-08-08 **)
ACTION Act_Link:

	IF tyMcParamCurr.eAGVComProtocol = McSetAGVCommOPCUA
		OR tyMcParamCurr.eAGVComProtocol = McSetAGVCommHardIO
		THEN
		IF tyMcParamCurr.eMagExMode = McSetMagXcAutoManMode
			OR tyMcParamCurr.eMagExMode = McSetMagXcAutoMode
			THEN
			tyMcParamCurr.bAGVComEn := TRUE;
		ELSE
			tyMcParamCurr.bAGVComEn := FALSE;
		END_IF
	ELSIF tyMcParamCurr.eAGVComProtocol = McSetAGVCommDisabled THEN
		tyMcParamCurr.bAGVComEn := FALSE;
	END_IF

	//new for Hermes 1.3
	IF p_bRmtHermesWriteConfig OR p_bSvyHermesWriteConfig THEN
		p_tyMcParamWr.sMcNm := p_tyHermesConfigurationWr.tySvyParam.sMachineId;
	END_IF

	//Disable MES on SMEMA mode
	IF p_eNtParamCustomerReq = Siemens AND tyMcParamCurr.eDSCommA <> McSetCommModHermes  AND ( NOT(p_bNtParamProjLaneBPrep) OR (p_bNtParamProjLaneBPrep AND tyMcParamCurr.eDSCommB <> McSetCommModHermes)) THEN
		tyMcParamCurr.bMesRFIDEn := FALSE;
		tyMcParamCurr.bHermesSvyEn := FALSE;
	END_IF
END_ACTION
```

#### Init.st
```iecst
(** 2019-05-04 **)
PROGRAM _INIT

	(* Always Change If Project Change *)

	//Pass Address To Global Address For External Use
	//Action, State & Status
	p_McParamStat		:= ADR(eStat);
	p_McParamStatus		:= ADR(eStatus);
	p_McParamStatTxt	:= ADR(sStatTxt);

	//Alarm
	p_McParamAlmData	:= ADR(tyAlmData);

	//Output
	p_McParamFileNotFound				:= ADR(bFileNotFound);

	p_McParamCurr						:= ADR(tyMcParamCurr);

	p_McParamLFOnline					:= ADR(tyMcParamCurr.a_bLFOnline);
	p_McParamLFIPAddr					:= ADR(tyMcParamCurr.a_sLFIPAddr);

	p_McParamMcNm						:= ADR(tyMcParamCurr.sMcNm);
	p_McParamSSaverTm					:= ADR(tyMcParamCurr.uiSSaverTmInSec);
	p_McParamSSaverEn					:= ADR(tyMcParamCurr.bSSaverEn);
	p_McParamDefaultMcMod				:= ADR(tyMcParamCurr.usiDefaultMcMod);
	p_McParamDefaultFlippedBrd			:= ADR(tyMcParamCurr.usiDefaultFlippedBrd);
	p_McParamWidthAtHmPos				:= ADR(tyMcParamCurr.diWidthAtHmPosInUM);
	p_McParamConvInitTm					:= ADR(tyMcParamCurr.diConvInitTmInMS);
	p_McParamTranOutErrDlyTm			:= ADR(tyMcParamCurr.diTranOutErrDlyTmInMS);
	p_McParamMag1ConvRunTmOut			:= ADR(tyMcParamCurr.diMag1ConvRunTmOutInMS);
	p_McParamMag2ConvRunTmOut			:= ADR(tyMcParamCurr.diMag2ConvRunTmOutInMS);
	p_McParamMag3ConvRunTmOut			:= ADR(tyMcParamCurr.diMag3ConvRunTmOutInMS);
	p_McParamMag4ConvRunTmOut			:= ADR(tyMcParamCurr.diMag4ConvRunTmOutInMS);
	p_McParamTravPosA					:= ADR(tyMcParamCurr.diTravPosA);
	p_McParamTravPosB					:= ADR(tyMcParamCurr.diTravPosB);
	p_McParamLifterPosA					:= ADR(tyMcParamCurr.diLifterPosA);
	p_McParamLifterPosB					:= ADR(tyMcParamCurr.diLifterPosB);
	p_McParamAWDis						:= ADR(tyMcParamCurr.bAWDis);
	p_McParamMnlAccDat					:= ADR(tyMcParamCurr.bMnlAccDat);
	p_McParamAutoStepEn					:= ADR(tyMcParamCurr.bAutoStepEn);
	p_McParamVSMEMAEn					:= ADR(tyMcParamCurr.bVSMEMAEn);
	p_McParamChgParamEn					:= ADR(tyMcParamCurr.bChgParamEn);
	p_McParamHermesRmtEn				:= ADR(tyMcParamCurr.bHermesRmtEn);
	p_McParamLongBrdEn					:= ADR(tyMcParamCurr.bLongBrdEn);
	p_McParamOutShutterDis				:= ADR(tyMcParamCurr.bOutShutterDis);
	p_McParamMagAutoDetTm				:= ADR(tyMcParamCurr.diMagAutoDetectSenTmInMS);
	p_McParamAGVComEn					:= ADR(tyMcParamCurr.bAGVComEn);

	p_McParamLFEn						:= ADR(tyMcParamCurr.bLFEn);
	p_McParamLCSLFEn					:= ADR(tyMcParamCurr.bLCSLFEn);
	p_McParamLCSReqRcpEn				:= ADR(tyMcParamCurr.bLCSReqRcpEn);
	p_McParamLCSManageRcpEn				:= ADR(tyMcParamCurr.bLCSManageRcpEn);
	p_McParamLCSLiveDatEn				:= ADR(tyMcParamCurr.bLCSLiveDatEn);
	p_McParamLFLeaderMc					:= ADR(tyMcParamCurr.bLFLeaderMc);
	p_McParamSectionLeader				:= ADR(tyMcParamCurr.bSectionLeader);
	p_McParamDSWidthChkEn				:= ADR(tyMcParamCurr.bDSWidthChkEn);
	p_McParamLFMcIdxBeforeOven			:= ADR(tyMcParamCurr.diLFMcIdxBeforeOven);
	p_McParamLFMcIdxAfterOven			:= ADR(tyMcParamCurr.diLFMcIdxAfterOven);

	p_McParamLang						:= ADR(tyMcParamCurr.usiLang);

	p_McParamConvLftSenAntiGap			:= ADR(tyMcParamCurr.tyLftSenAntiGapDly);
	p_McParamConvLftSenOnTm				:= ADR(tyMcParamCurr.tyLftSenAntiGapDly.diSigOnTm);
	p_McParamConvLftSenOffTm			:= ADR(tyMcParamCurr.tyLftSenAntiGapDly.diSigOffTm);
	p_McParamConvRgtSenAntiGap			:= ADR(tyMcParamCurr.tyRgtSenAntiGapDly);
	p_McParamConvRgtSenOnTm				:= ADR(tyMcParamCurr.tyRgtSenAntiGapDly.diSigOnTm);
	p_McParamConvRgtSenOffTm			:= ADR(tyMcParamCurr.tyRgtSenAntiGapDly.diSigOffTm);

	p_McParamMagConvEntrySenAntiGap		:= ADR(tyMcParamCurr.tyMagConvEntrySenAntiGapDly);
	p_McParamMagConvEntrySenOnTm		:= ADR(tyMcParamCurr.tyMagConvEntrySenAntiGapDly.diSigOnTm);
	p_McParamMagConvEntrySenOffTm		:= ADR(tyMcParamCurr.tyMagConvEntrySenAntiGapDly.diSigOffTm);

	p_McParamMagConvPresentAntiGap		:= ADR(tyMcParamCurr.tyMagConvPresentSenAntiGapDly);
	p_McParamMagConvPresentSenOnTm		:= ADR(tyMcParamCurr.tyMagConvPresentSenAntiGapDly.diSigOnTm);
	p_McParamMagConvPresentSenOffTm		:= ADR(tyMcParamCurr.tyMagConvPresentSenAntiGapDly.diSigOffTm);

	p_McParamDSCommAMod					:= ADR(tyMcParamCurr.eDSCommA);
	p_McParamDSSMEMAAParam				:= ADR(tyMcParamCurr.tyDSCommASMEMA);
	p_McParamDSSMEMAASelection			:= ADR(tyMcParamCurr.tyDSCommASMEMA.eSelection);
	p_McParamDBAAStatSetGd				:= ADR(tyMcParamCurr.tyDSCommASMEMA.bStatSigSetGd);

	p_McParamDSCommBMod					:= ADR(tyMcParamCurr.eDSCommB);
	p_McParamDSSMEMABParam				:= ADR(tyMcParamCurr.tyDSCommBSMEMA);
	p_McParamDSSMEMABSelection			:= ADR(tyMcParamCurr.tyDSCommBSMEMA.eSelection);
	p_McParamDBABStatSetGd				:= ADR(tyMcParamCurr.tyDSCommBSMEMA.bStatSigSetGd);

	p_McParamLFMcIdxBeforeOven2			:= ADR(tyMcParamCurr.diLFMcIdxBeforeOven2);
	p_McParamLFMcIdxAfterOven2			:= ADR(tyMcParamCurr.diLFMcIdxAfterOven2);
//	p_McParamAIVComm					:= ADR(tyMcParamCurr.tyAIVComm);
//	p_McParamAIVSvrPort					:= ADR(tyMcParamCurr.tyAIVComm.uiSvrPort);
//	p_McParamAIVClientPort				:= ADR(tyMcParamCurr.tyAIVComm.uiClientPort);
//	p_McParamAIVClientAddr				:= ADR(tyMcParamCurr.tyAIVComm.sClientAddress);

	p_McParamWidthOffset				:= ADR(tyMcParamCurr.diWidthOffsetInUM);

	p_McParamNetworkMod					:= ADR(tyMcParamCurr.eNetworkMod);

	p_McParamLFSeqStayActive			:= ADR(tyMcParamCurr.bLFSeqStayActive);
	p_McParamLFBuzMute					:= ADR(tyMcParamCurr.bLFBuzMute);

	p_McParamVID			     		:= ADR(tyMcParamCurr.diVID);
	p_McParamPID			    		:= ADR(tyMcParamCurr.diPID);
	p_McParamScannerEn					:= ADR(tyMcParamCurr.bScannerEn);

	p_McParamAGVComProtocol				:= ADR(tyMcParamCurr.eAGVComProtocol);
	p_McParamMagExMode					:= ADR(tyMcParamCurr.eMagExMode);

	p_McParamRS232StartCode1		:= ADR(tyMcParamCurr.diRS232StartCode1);
	p_McParamRS232StartCode2		:= ADR(tyMcParamCurr.diRS232StartCode2);
	p_McParamRS232EndCode1			:= ADR(tyMcParamCurr.diRS232EndCode1);
	p_McParamRS232EndCode2			:= ADR(tyMcParamCurr.diRS232EndCode2);

	p_McParamAWPusherAtHmPos			:= ADR(tyMcParamCurr.diAWPusherAtHmPosInUM);
	p_McParamAWPusherDis				:= ADR(tyMcParamCurr.bAWPusherDis);

	p_McParamTravOutletFixtoFixPos	:= ADR(tyMcParamCurr.diTravOutletFixtoFixPos);
	p_McParamDisableFMWarning		:= ADR(tyMcParamCurr.bDisableFMWarning);
	p_McParamDBAOnWOAlign			:= ADR(tyMcParamCurr.bDBAOnWOAlign);

	p_McParamMagWidthChkDis			:= ADR(tyMcParamCurr.bMagWidthChkDis);
	p_McParamMag1WidthChkDetDist	:= ADR(tyMcParamCurr.diMag1WidthChkDetDist);
	p_McParamMag2WidthChkDetDist	:= ADR(tyMcParamCurr.diMag2WidthChkDetDist);
	p_McParamMag3WidthChkDetDist	:= ADR(tyMcParamCurr.diMag3WidthChkDetDist);
	p_McParamDBAOnRgtSen 		    := ADR(tyMcParamCurr.bDBAOnRgtSen);						    // ADD for OPL 52: Shift bDBAOnRgtSen frm NtParam to Mc Param
	p_McParamHermesSvyEn			:= ADR(tyMcParamCurr.bHermesSvyEn);//new for Hermes 1.3
	p_McParamHermesScannerEn		:= ADR(tyMcParamCurr.bHermesScannerEn);//new for Hermes 1.3
	p_McParamMesRFIDEn				:= ADR(tyMcParamCurr.bMesRFIDEn);
	p_McParamMesRFIDTOInMS			:= ADR(tyMcParamCurr.diMesRFIDTOInMS);
	p_McParamTravLaneBOffset		:= ADR(tyMcParamCurr.diTravLaneBOffset);

	(* Always Change If Project Change *)

END_PROGRAM
```

### NtParam.typ
```iecst
(*2022-03-15 (note for diProjMagMaxSlt and diProjPullerExtMaxSlt)*)
(**)
(*Action*)

TYPE
	eNtParamAction :
		(
		NtParamActIdle,
		NtParamActCreateDir,
		NtParamActRead,
		NtParamActWrite,
		NtParamActLoad,
		NtParamActSave
		);
END_TYPE

(**)
(*Data*)

TYPE
	tyNtParam : 	STRUCT
		tyDISettings : tyDigitalInputSettings := (diSafetyRlySig:=1,diEStopSig:=2,diCoverSWSig:=3,diDSBA:=4,diDSBB:=5,diPullerExtRS:=8,diPullerRetRS:=9,diPullerRotHmRS:=47,diPullerRotRmRS:=48,diConvLftSen:=12,diConvRgtSen:=13,diLifterTimingBeltSen:=16,diLifterSafetyLmtSW1:=0,diLifterSafetyLmtSW2:=0,diMag1FixedClampRS:=35,diMag1FixedUnclampRS:=32,diMag1RemoteClampRS:=0,diMag1RemoteUnclampRS:=64,diMag2FixedClampRS:=36,diMag2FixedUnclampRS:=33,diMag2RemoteClampRS:=0,diMag2RemoteUnclampRS:=65,diMag3FixedClampRS:=37,diMag3FixedUnclampRS:=34,diMag3RemoteClampRS:=0,diMag3RemoteUnclampRS:=66,diMag4FixedClampRS:=0,diMag4FixedUnclampRS:=0,diMag4RemoteClampRS:=0,diMag4RemoteUnclampRS:=0,diInShutterOpenRS:=21,diInShutterCloseRS:=22,diOutShutterOpenRS:=23,diOutShutterCloseRS:=24,diMagPresentSen1:=17,diMagPresentSen2:=18,diMagPresentSen3:=19,diMagPresentSen4:=0,diMagConvEntSen1:=29,diMagConvEntSen2:=30,diMagConvEntSen3:=31,diMagConvEntSen4:=0,diMag1AGVInPosSen1:=0,diMag1AGVInPosSen2:=0,diMag2AGVInPosSen1:=0,diMag2AGVInPosSen2:=0,diMag3AGVInPosSen1:=0,diMag3AGVInPosSen2:=0,diMag4AGVInPosSen1:=0,diMag4AGVInPosSen2:=0,diMag1OrientChkSen1:=42,diMag1OrientChkSen2:=0,diMag2OrientChkSen1:=43,diMag2OrientChkSen2:=0,diMag3OrientChkSen1:=44,diMag3OrientChkSen2:=0,diMag4OrientChkSen1:=0,diMag4OrientChkSen2:=0,diDSWidthChkSen:=0,diMagConvHeightSen1:=68,diMagConvHeightSen2:=70,diMagConvHeightSen3:=72,diMagConvHeightSen4:=0,diMagConvSmallMagSen1:=0,diMagConvSmallMagSen2:=0,diMagConvSmallMagSen3:=0,diMagConvSmallMagSen4:=0,diMagConvLargeMagSen1:=0,diMagConvLargeMagSen2:=0,diMagConvLargeMagSen3:=0,diMagConvLargeMagSen4:=0,diMagConvCAB717MagSen1:=0,diMagConvCAB717MagSen2:=0,diMagConvCAB717MagSen3:=0,diMagConvCAB717MagSen4:=0,diMag1SelUnClampRS:=0,diMag2SelUnClampRS:=0,diMag3SelUnClampRS:=0,diMag4SelUnClampRS:=0,diSOT1Receive:=53,diSOT1AIVError:=49,diSOT1AIVSizeLarge:=50,diSOT1AIVReady:=51,diSOT1AIVAvailable:=52,diSOT2Receive:=58,diSOT2AIVError:=54,diSOT2AIVSizeLarge:=55,diSOT2AIVReady:=56,diSOT2AIVAvailable:=57,diSOT3Receive:=63,diSOT3AIVError:=59,diSOT3AIVSizeLarge:=60,diSOT3AIVReady:=61,diSOT3AIVAvailable:=62,diSOT4Receive:=0,diSOT4AIVError:=0,diSOT4AIVSizeLarge:=0,diSOT4AIVReady:=0,diSOT4AIVAvailable:=0,diFleetManagerReady:=0,diPullerExtSlwSen:=38,diPullerRetSlwSen:=39,diMtrPullerTorqueSig:=0,diMtrPullerAlmSig:=0,diMag1SafetyBarExtRS:=0,diMag1SafetyBarRetRS:=0,diMag2SafetyBarExtRS:=0,diMag2SafetyBarRetRS:=0,diMag3SafetyBarExtRS:=0,diMag3SafetyBarRetRS:=0,diMag4SafetyBarExtRS:=0,diMag4SafetyBarRetRS:=0,diMagWidthChkSen:=45,diPullerAntiJam:=0,diCurtainSensor:=20,diBypCurtainSensorPB:=46,diInShutterOpenRS2:=25,diInShutterCloseRS2:=26,diInShutterOpenRS3:=27,diInShutterCloseRS3:=28,diMag1FixedSideDetect:=67,diMag1RemoteSideDetect:=0,diMag2FixedSideDetect:=69,diMag2RemoteSideDetect:=0,diMag3FixedSideDetect:=71,diMag3RemoteSideDetect:=0,diCurtainSafetySig2:=40,diHighMagDetSen1:=0,diHighMagDetSen2:=0,diHighMagDetSen3:=0,diConvClrSen:=14,diDSUnlockCoverSig:=0,diDSSafetySig:=0,diOutShutterOpenRS2:=0,diOutShutterCloseRS2:=0,diTrolleyExtRS1:=0,diTrolleyExtRS2:=0,diTrolleyPreSen1:=0,diTrolleyPreSen2:=0,diSlotLckSenMag1:=0,diSlotLckSenMag2:=0,diSPARE16:=0,diSPARE17:=0,diSPARE18:=0,diSPARE19:=0,diSPARE20:=0);
		tyDOSettings : tyDigitalOutputSettings := (diSafetyRlyRst:=1,diTLRed:=4,diTLAmber:=3,diTLGreen:=2,diBuzzer:=5,diDBAA:=8,diDBAB:=9,diPullerExtCtrl:=0,diPullerRetCtrl:=0,diRotPullerCtrl:=13,diMag1FixedClampCtrl:=23,diMag1RemoteClampCtrl:=26,diMag2FixedClampCtrl:=24,diMag2RemoteClampCtrl:=27,diMag3FixedClampCtrl:=25,diMag3RemoteClampCtrl:=28,diMag4FixedClampCtrl:=0,diMag4RemoteClampCtrl:=0,diInShutterOpenCtrl:=17,diInShutterCloseCtrl:=18,diOutShutterOpenCtrl:=15,diOutShutterCloseCtrl:=16,diMag1ConvMtrIn:=31,diMag1ConvMtrOut:=32,diMag2ConvMtrIn:=33,diMag2ConvMtrOut:=34,diMag3ConvMtrIn:=35,diMag3ConvMtrOut:=36,diMag4ConvMtrIn:=0,diMag4ConvMtrOut:=0,diPullConvMtrOn:=14,diMag1SelClampCtrl:=0,diMag2SelClampCtrl:=0,diMag3SelClampCtrl:=0,diMag4SelClampCtrl:=0,diSOT1MagError:=43,diSOT1MagSizeLarge:=44,diSOT1MagReady:=45,diSOT1MagAvailable:=46,diSOT2MagError:=47,diSOT2MagSizeLarge:=48,diSOT2MagReady:=49,diSOT2MagAvailable:=50,diSOT3MagError:=51,diSOT3MagSizeLarge:=52,diSOT3MagReady:=53,diSOT3MagAvailable:=54,diSOT4MagError:=0,diSOT4MagSizeLarge:=0,diSOT4MagReady:=0,diSOT4MagAvailable:=0,diMag1ReqToBring:=0,diMag1ReqToGet:=0,diMag2ReqToBring:=0,diMag2ReqToGet:=0,diMag3ReqToBring:=0,diMag3ReqToGet:=0,diMag4ReqToBring:=0,diMag4ReqToGet:=0,diUSBRun:=0,diMtrPshrExt:=0,diMtrPshrRet:=0,diMtrPshrOn:=0,diMtrPshrBrakeRls:=0,diMtrPshrSpdBinBit0:=0,diMtrPshrSpdBinBit1:=0,diMtrPshrSpdBinBit2:=0,diMtrPshrAlmRst:=0,diMag1SafetyBarRetCtrl:=0,diMag2SafetyBarRetCtrl:=0,diMag3SafetyBarRetCtrl:=0,diBypCurtainSen:=39,diBypCurtainSensorPBLED:=6,diRstCurtainSen:=40,diInShutterOpenCtrl2:=19,diInShutterCloseCtrl2:=20,diInShutterOpenCtrl3:=21,diInShutterCloseCtrl3:=22,diMag1FixedClampOpenCtrl:=29,diMag1RemoteClampOpenCtrl:=38,diMag2FixedClampOpenCtrl:=30,diMag2RemoteClampOpenCtrl:=41,diMag3FixedClampOpenCtrl:=37,diMag3RemoteClampOpenCtrl:=42,diMag4FixedClampOpenCtrl:=0,diMag4RemoteClampOpenCtrl:=0,diMcSafetySigToDS:=0,diOutShutterOpenCtrl2:=0,diOutShutterCloseCtrl2:=0,diTrolleyLckCtrl1:=0,diTrolleyLckCtrl2:=0,diSPARE15:=0,diSPARE16:=0,diSPARE17:=0,diSPARE18:=0,diSPARE19:=0,diSPARE20:=0);
		bAWPusherPrep : BOOL := TRUE;
		bAWPrep : BOOL := TRUE;
		bLFPrep : BOOL := TRUE;
		bLeaderMc : BOOL := TRUE;
		bLFUsrSetPrep : BOOL := TRUE;
		diLFWidthLimit : DINT := 3000;
		bLFProdWidthChk : BOOL := FALSE;
		bDSWidthChkPrep : BOOL := FALSE;
		bLCSLFPrep : BOOL := FALSE;
		bLCSReqRcpPrep : BOOL := FALSE;
		bLCSManageRcpPrep : BOOL := FALSE;
		bLCSLiveDatPrep : BOOL := FALSE;
		bIPCSMEMA9851ExtdPrep : BOOL := FALSE;
		bVSMEMAPrep : BOOL := TRUE;
		bHermesPrep : BOOL := TRUE;
		bHermesRmtPrep : BOOL := TRUE;
		bSSaverPrep : BOOL := TRUE;
		diAWPushPulOffsetInUM : DINT := 0;
		diWidthOffsetInUM : DINT := 0;
		sJobNo : STRING[30] := '2023-0301P01';
		usiNtAddr : USINT := 4;
		bProjLifterMagPlatform : BOOL := FALSE;
		bProjLaneBPrep : BOOL := FALSE;
		bProjTopToBtmDefault : BOOL := FALSE;
		bProjLongBrdPrep : BOOL := FALSE;
		bProjInletShutPrep : BOOL := TRUE;
		bProjOutletShutPrep : BOOL := TRUE;
		bProjMag1ConvPrep : BOOL := TRUE;
		bProjMag2ConvPrep : BOOL := TRUE;
		bProjMag3ConvPrep : BOOL := TRUE;
		bProjMag4ConvPrep : BOOL := FALSE;
		bProjMagOrientChkSenPrep : BOOL := TRUE;
		bProjAGVPrep : BOOL := TRUE;
		bProjAGVInPosSenPrep : BOOL := FALSE;
		bProjBypsInitConvPrep : BOOL := TRUE;
		bProjRlsNewProdPrep : BOOL := FALSE;
		bProjBtnInsertRmvMag : BOOL := TRUE;
		bProjSOTSensorPrep : BOOL := FALSE;
		bProjMotorizedPullerPrep : BOOL := TRUE;
		bProjMagSafetyBarPrep : BOOL := FALSE;
		diProjMagMinSlt : DINT := 5;
		diProjMagMaxSlt : DINT := 60;
		eProjMag : eLDMag := LDMagTriple;
		eProjConvDir : eConvDir := ConvDirLToR;
		eProjMagConvDir : eConvDir := ConvDirLToL;
		sUsrFolderProgNm : STRING[15] := 'UsrFolder';
		sLibVersionProgNm : STRING[15] := 'LibVer';
		sTimeProgNm : STRING[15] := 'Time';
		sHWInfoProgNm : STRING[15] := 'HWInfo';
		sHWInfoDevice : STRING[3] := 'IF2';
		tTLChgRcpBlinkTm : TIME := T#500ms;
		tTLErrBlinkTm : TIME := T#500ms;
		tBuzErrOnTm : TIME := T#500ms;
		tBuzErrRestTm : TIME := T#500ms;
		usiBuzErrOnCntr : USINT := 3;
		bBuzErrStopSeqEn : BOOL := FALSE;
		usiBuzErrStopSeqCntr : USINT := 3;
		tTLWarnBlinkTm : TIME := T#500ms;
		tBuzWarnOnTm : TIME := T#500ms;
		tBuzWarnRestTm : TIME := T#5s;
		usiBuzWarnOnCntr : USINT := 3;
		bBuzWarnStopSeqEn : BOOL := FALSE;
		usiBuzWarnStopSeqCntr : USINT := 3;
		tTLWarn1BlinkTm : TIME := T#500ms;
		tBuzWarn1OnTm : TIME := T#500ms;
		tBuzWarn1RestTm : TIME := T#5s;
		usiBuzWarn1OnCntr : USINT := 3;
		bBuzWarn1StopSeqEn : BOOL := FALSE;
		usiBuzWarn1StopSeqCntr : USINT := 3;
		tTLWarn2BlinkTm : TIME := T#500ms;
		tBuzWarn2OnTm : TIME := T#500ms;
		tBuzWarn2RestTm : TIME := T#5s;
		usiBuzWarn2OnCntr : USINT := 3;
		bBuzWarn2StopSeqEn : BOOL := FALSE;
		usiBuzWarn2StopSeqCntr : USINT := 3;
		tTLWarn3BlinkTm : TIME := T#500ms;
		tBuzWarn3OnTm : TIME := T#500ms;
		tBuzWarn3RestTm : TIME := T#5s;
		usiBuzWarn3OnCntr : USINT := 3;
		bBuzWarn3StopSeqEn : BOOL := FALSE;
		usiBuzWarn3StopSeqCntr : USINT := 3;
		tTLWarn4BlinkTm : TIME := T#500ms;
		tBuzWarn4OnTm : TIME := T#500ms;
		tBuzWarn4RestTm : TIME := T#5s;
		usiBuzWarn4OnCntr : USINT := 3;
		bBuzWarn4StopSeqEn : BOOL := FALSE;
		usiBuzWarn4StopSeqCntr : USINT := 3;
		tTLWarn5BlinkTm : TIME := T#500ms;
		tBuzWarn5OnTm : TIME := T#500ms;
		tBuzWarn5RestTm : TIME := T#5s;
		usiBuzWarn5OnCntr : USINT := 3;
		bBuzWarn5StopSeqEn : BOOL := FALSE;
		usiBuzWarn5StopSeqCntr : USINT := 3;
		tBuzAlertOnTm : TIME := T#500ms;
		tBuzAlertRestTm : TIME := T#5s;
		usiBuzAlertOnCntr : USINT := 3;
		bBuzAlertStopSeqEn : BOOL := FALSE;
		usiBuzAlertStopSeqCntr : USINT := 3;
		tTLBlueBlinkTm : TIME := T#500ms;
		tTLAmberBlinkTm : TIME := T#500ms;
		tTLWhiteBlinkTm : TIME := T#500ms;
		tTLRedBlinkTm : TIME := T#500ms;
		tTLGreenBlinkTm : TIME := T#500ms;
		eTLBuzMode : eTLBuzMod := TLBuzModNutek;
		sAlmProgNm : STRING[15] := 'Alarm';
		udiAlmFileKeepDay : UDINT := 30;
		sProdRcpProgNm : STRING[15] := 'ProdRcp';
		sProdRcpListFileNm : STRING[80] := 'ProductRecipeList.dat';
		sProdRcpSingleFileNm : STRING[80] := 'ProductRecipe.dat';
		sMpProdRcpProgNm : STRING[15] := 'MpProdRcp';
		sMpProdRcpFileNm : STRING[255] := 'MpProductRecipe.xml';
		sMpProdRcpPVNm : STRING[100] := 'MpProdRcp:a_tyMpProdRcp1';
		sMagRcpProgNm : STRING[15] := 'MagRcp';
		sMagRcpListFileNm : STRING[80] := 'MagazineRecipeList.dat';
		sMagRcpSingleFileNm : STRING[80] := 'MagazineRecipe.dat';
		sMagRcpProgNm1 : STRING[15] := 'MagRcp1';
		sMagRcpListFileNm1 : STRING[80] := 'MagazineRecipeList1.dat';
		sMagRcpSingleFileNm1 : STRING[80] := 'MagazineRecipe1.dat';
		sMcParamProgNm : STRING[15] := 'McParam';
		sMcParamFileNm : STRING[80] := 'MachineParameter.dat';
		sUsrMgmtProgNm : STRING[15] := 'UsrMgmt';
		sBffr1ProgNm : STRING[15] := 'Buffer 1';
		sBffr1FileNm : STRING[80] := 'Buffer1.dat';
		bBffr1FIFO : BOOL := TRUE;
		sBffr2ProgNm : STRING[15] := 'Buffer 2';
		sBffr2FileNm : STRING[80] := 'Buffer2.dat';
		bBffr2FIFO : BOOL := TRUE;
		sBffr3ProgNm : STRING[15] := 'Buffer 3';
		sBffr3FileNm : STRING[80] := 'Buffer3.dat';
		bBffr3FIFO : BOOL := TRUE;
		sBffr4ProgNm : STRING[15] := 'Buffer 4';
		sBffr4FileNm : STRING[80] := 'Buffer4.dat';
		bBffr4FIFO : BOOL := TRUE;
		sUSSMEMA1ProgNm : STRING[15] := 'Mag1_US';
		tUSSMEMA1RstDlyTm : TIME := T#0s;
		tUSSMEMA1SigInChkTm : TIME := T#100ms;
		sUSSMEMA2ProgNm : STRING[15] := 'Mag2_US';
		tUSSMEMA2RstDlyTm : TIME := T#0s;
		tUSSMEMA2SigInChkTm : TIME := T#100ms;
		sUSSMEMA3ProgNm : STRING[15] := 'Mag3_US';
		tUSSMEMA3RstDlyTm : TIME := T#0s;
		tUSSMEMA3SigInChkTm : TIME := T#100ms;
		sUSSMEMA4ProgNm : STRING[15] := 'Mag4_US';
		tUSSMEMA4RstDlyTm : TIME := T#0s;
		tUSSMEMA4SigInChkTm : TIME := T#100ms;
		sDSSMEMA1ProgNm : STRING[15] := 'Mag1_DS';
		tDSSMEMA1RstDlyTm : TIME := T#0s;
		tDSSMEMA1SigInChkTm : TIME := T#100ms;
		sDSSMEMA2ProgNm : STRING[15] := 'Mag2_DS';
		tDSSMEMA2RstDlyTm : TIME := T#0s;
		tDSSMEMA2SigInChkTm : TIME := T#100ms;
		sDSSMEMA3ProgNm : STRING[15] := 'Mag3_DS';
		tDSSMEMA3RstDlyTm : TIME := T#0s;
		tDSSMEMA3SigInChkTm : TIME := T#100ms;
		sDSSMEMA4ProgNm : STRING[15] := 'Mag4_DS';
		tDSSMEMA4RstDlyTm : TIME := T#0s;
		tDSSMEMA4SigInChkTm : TIME := T#100ms;
		sDSSMEMAAProgNm : STRING[15] := 'DSSMEMA A';
		tDSSMEMAARstDlyTm : TIME := T#500ms;
		tDSSMEMAASigInChkTm : TIME := T#100ms;
		sDSSMEMABProgNm : STRING[15] := 'DSSMEMA B';
		tDSSMEMABRstDlyTm : TIME := T#500ms;
		tDSSMEMABSigInChkTm : TIME := T#100ms;
		sInShutterProgNm : STRING[15] := 'Inlet Shutter';
		bInShutterTwoCtrlIn : BOOL := TRUE;
		tInShutterExtTO : TIME := T#20s;
		tInShutterRetTO : TIME := T#20s;
		sOutShutterProgNm : STRING[15] := 'Outlet Shutter';
		bOutShutterTwoCtrlIn : BOOL := TRUE;
		tOutShutterExtTO : TIME := T#20s;
		tOutShutterRetTO : TIME := T#20s;
		sSelClamp1ProgNm : STRING[15] := 'Sel Clamp 1';
		bSelClamp1TwoCtrlIn : BOOL := FALSE;
		tSelClamp1ExtDlyTm : TIME := T#10s;
		tSelClamp1RetDlyTm : TIME := T#10s;
		sSelClamp2ProgNm : STRING[15] := 'Sel Clamp 2';
		bSelClamp2TwoCtrlIn : BOOL := FALSE;
		tSelClamp2ExtDlyTm : TIME := T#10s;
		tSelClamp2RetDlyTm : TIME := T#10s;
		sSelClamp3ProgNm : STRING[15] := 'Sel Clamp 3';
		bSelClamp3TwoCtrlIn : BOOL := FALSE;
		tSelClamp3ExtDlyTm : TIME := T#10s;
		tSelClamp3RetDlyTm : TIME := T#10s;
		sSelClamp4ProgNm : STRING[15] := 'Sel Clamp 4';
		bSelClamp4TwoCtrlIn : BOOL := FALSE;
		tSelClamp4ExtDlyTm : TIME := T#10s;
		tSelClamp4RetDlyTm : TIME := T#10s;
		sMag1SafetyBarProgNm : STRING[15] := 'Mag1 SafetyBar';
		bMag1SafetyBarTwoCtrlIn : BOOL := FALSE;
		tMag1SafetyBarExtTO : TIME := T#20s;
		tMag1SafetyBarRetTO : TIME := T#20s;
		sMag2SafetyBarProgNm : STRING[15] := 'Mag2 SafetyBar';
		bMag2SafetyBarTwoCtrlIn : BOOL := FALSE;
		tMag2SafetyBarExtTO : TIME := T#20s;
		tMag2SafetyBarRetTO : TIME := T#20s;
		sMag3SafetyBarProgNm : STRING[15] := 'Mag3 SafetyBar';
		bMag3SafetyBarTwoCtrlIn : BOOL := FALSE;
		tMag3SafetyBarExtTO : TIME := T#20s;
		tMag3SafetyBarRetTO : TIME := T#20s;
		sMag4SafetyBarProgNm : STRING[15] := 'Mag4 SafetyBar';
		bMag4SafetyBarTwoCtrlIn : BOOL := FALSE;
		tMag4SafetyBarExtTO : TIME := T#20s;
		tMag4SafetyBarRetTO : TIME := T#20s;
		sPullConvProgNm : STRING[15] := 'PullerConv';
		bPullConvOnDirMod : BOOL := FALSE;
		tPullConvMtrOffDlyTm : TIME := T#0s;
		tPullConvPullExtTO : TIME := T#20s;
		tPullConvPullRetTO : TIME := T#20s;
		tPullConvRotHomeTO : TIME := T#20s;
		tPullConvRotRemoteTO : TIME := T#20s;
		sMagConv1ProgNm : STRING[15] := 'MagConv 1';
		bMagConv1OnDirMod : BOOL := FALSE;
		tMagConv1MtrOffDlyTm : TIME := T#0s;
		tMagConv1ClprClampTO : TIME := T#20s;
		tMagConv1ClprUnclampTO : TIME := T#20s;
		sMagConv2ProgNm : STRING[15] := 'MagConv 2';
		bMagConv2OnDirMod : BOOL := FALSE;
		tMagConv2MtrOffDlyTm : TIME := T#0s;
		tMagConv2ClprClampTO : TIME := T#20s;
		tMagConv2ClprUnclampTO : TIME := T#20s;
		sMagConv3ProgNm : STRING[15] := 'MagConv 3';
		bMagConv3OnDirMod : BOOL := FALSE;
		tMagConv3MtrOffDlyTm : TIME := T#0s;
		tMagConv3ClprClampTO : TIME := T#20s;
		tMagConv3ClprUnclampTO : TIME := T#20s;
		sMagConv4ProgNm : STRING[15] := 'MagConv 4';
		bMagConv4OnDirMod : BOOL := FALSE;
		tMagConv4MtrOffDlyTm : TIME := T#0s;
		tMagConv4ClprClampTO : TIME := T#20s;
		tMagConv4ClprUnclampTO : TIME := T#20s;
		sMtrPshrProgNm : STRING[15] := 'MotorizedPuller';
		bMtrPshrDir : BOOL := TRUE;
		tMtrPshrAlmRstTm : TIME := T#1s;
		tMtrPshrAlmTrigTm : TIME := T#1s;
		tMtrPshrExtTO : TIME := T#20s;
		tMtrPshrRetTO : TIME := T#20s;
		diMtrPshrExtSlowSpd : DINT := 1;
		diMtrPshrRetSlowSpd : DINT := 1;
		diMtrPshrExtNomSpd : DINT := 8;
		diMtrPshrExtTorq : DINT := 40;
		diMtrPshrRetTorq : DINT := 50;
		diMtrPshrStartTorq : DINT := 90;
		sAWPushPullProgNm : STRING[15] := 'AWPuller';
		sAWPushPullDevice : STRING[3] := 'IF7';
		usiAWPushPullNode : USINT := 19;
		bAWPushPullDir : BOOL := FALSE;
		bAWPushPullDirBl : BOOL := FALSE;
		diAWPushPullPitchInUM : DINT := 3000;
		diAWPushPullMovBlDistInUM : DINT := 3000;
		tyAWPushPullParamInHm : tyMotionCANParamInHm := (diStartVelInUMPS:=10000,diAcc:=50);
		tyAWPushPullParamInConvert : tyMotionCANParamInConvert := (diPitchInUM:=3000);
		tyAWPushPullParam : tyMotionParam := (diAccInMS:=500,diDecInMS:=500,diAutoSpdInUMPS:=15000);
		tyAWPushPullTuning : tyMotionCANTuning := (diAsdaA2Inertia:=76,diAsdaA2PosLoopGain:=53,diAsdaA2PosFFGain:=50,diAsdaA2SpdLoopGain:=213,diAsdaA2SpdIntegral:=34,diAsdaA2LowPassFltr:=49,diAsdaA2AntiInterGain:=34,diAsdaA2FirstTorqueCmd:=300,diLex28LTNDderivativeGain_P800:=0,diLex28LTNIintegralGain_P801:=0,diLex28LTNIVdeIntlGain_P802:=0,diLex28LTNPpropotionalGain_P803:=0,diLex28LTNUSERGAIN_P804:=0,diLex28NLAFFLPFHZspringFil_P805:=0,diLex28NLFILTDAMPING_P814:=0,diLex28NLFILTT1_P815:=0,diPronetInertia:=100,diPronetRealTimeAutoAdjSet:=0,diPronetPosLoopGain:=40,diPronetSpdLoopGain:=250,diPronetSpdIntegral:=200,diPronetTorqueFilter:=100,diPronetPosFeedForward:=0,diPronetLowSpeedTestFiltering:=10,diPronetStopMode:=5);
		eAWPushPullServoMotorType : eServoMotorType := DeltaAsdaA2; (*Selection of  Motor Brand*)
		sAWProgNm : STRING[15] := 'AWOpen';
		sAWDevice : STRING[3] := 'IF7';
		usiAWNode : USINT := 16;
		bAWDir : BOOL := TRUE;
		bAWDirBl : BOOL := FALSE;
		diAWPitchInUM : DINT := 3000;
		diAWMovBlDistInUM : DINT := 3000;
		tyAWParamInHm : tyMotionCANParamInHm := (diStartVelInUMPS:=15000,diAcc:=25);
		tyAWParamInConvert : tyMotionCANParamInConvert := (diPitchInUM:=3000); (*estun1048576*)
		tyAWParam : tyMotionParam := (diAccInMS:=500,diDecInMS:=500,diAutoSpdInUMPS:=15000);
		tyAWTuning : tyMotionCANTuning := (diAsdaA2Inertia:=76,diAsdaA2PosLoopGain:=53,diAsdaA2PosFFGain:=50,diAsdaA2SpdLoopGain:=213,diAsdaA2SpdIntegral:=34,diAsdaA2LowPassFltr:=49,diAsdaA2AntiInterGain:=34,diAsdaA2FirstTorqueCmd:=300,diLex28LTNDderivativeGain_P800:=0,diLex28LTNIintegralGain_P801:=0,diLex28LTNIVdeIntlGain_P802:=0,diLex28LTNPpropotionalGain_P803:=0,diLex28LTNUSERGAIN_P804:=0,diLex28NLAFFLPFHZspringFil_P805:=0,diLex28NLFILTDAMPING_P814:=0,diLex28NLFILTT1_P815:=0,diPronetInertia:=0,diPronetRealTimeAutoAdjSet:=0,diPronetPosLoopGain:=80,diPronetSpdLoopGain:=750,diPronetSpdIntegral:=600,diPronetTorqueFilter:=4,diPronetPosFeedForward:=0,diPronetLowSpeedTestFiltering:=0,diPronetStopMode:=5);
		eAWServoMotorType : eServoMotorType := DeltaAsdaA2; (*Selection of  Motor Brand*)
		sTravProgNm : STRING[15] := 'Trav';
		sTravDevice : STRING[3] := 'IF7';
		usiTravNode : USINT := 18;
		bTravDir : BOOL := FALSE;
		tyTravParamInHm : tyMotionCANParamInHm := (diStartVelInUMPS:=50000,diAcc:=25);
		tyTravParamInConvert : tyMotionCANParamInConvert := (diPitchInUM:=190530,diPrimaryGearRatio:=1,diSecondaryGearRatio:=10); (*belt190530*)
		tyTravParam : tyMotionParam := (diAccInMS:=500,diDecInMS:=500,diAutoSpdInUMPS:=100000);
		tyTravTuning : tyMotionCANTuning := (diAsdaA2Inertia:=76,diAsdaA2PosLoopGain:=53,diAsdaA2PosFFGain:=50,diAsdaA2SpdLoopGain:=213,diAsdaA2SpdIntegral:=34,diAsdaA2LowPassFltr:=49,diAsdaA2AntiInterGain:=34,diAsdaA2FirstTorqueCmd:=300,diLex28LTNDderivativeGain_P800:=0,diLex28LTNIintegralGain_P801:=0,diLex28LTNIVdeIntlGain_P802:=0,diLex28LTNPpropotionalGain_P803:=0,diLex28LTNUSERGAIN_P804:=0,diLex28NLAFFLPFHZspringFil_P805:=0,diLex28NLFILTDAMPING_P814:=0,diLex28NLFILTT1_P815:=0,diPronetInertia:=0,diPronetRealTimeAutoAdjSet:=0,diPronetPosLoopGain:=20,diPronetSpdLoopGain:=450,diPronetSpdIntegral:=400,diPronetTorqueFilter:=4,diPronetPosFeedForward:=0,diPronetLowSpeedTestFiltering:=0,diPronetStopMode:=5);
		eTravServoMotorType : eServoMotorType := DeltaAsdaA2; (*Selection of  Motor Brand*)
		diTravAutoSpdLongBrdInUMPS : DINT := 100000;
		sLifterProgNm : STRING[15] := 'LifterBtm';
		sLifterDevice : STRING[3] := 'IF7';
		usiLifterNode : USINT := 17;
		bLifterDir : BOOL := TRUE;
		tyLifterParamInHm : tyMotionCANParamInHm := (diStartVelInUMPS:=25000,diAcc:=25);
		tyLifterParamInConvert : tyMotionCANParamInConvert := (diPitchInUM:=10000);
		tyLifterParam : tyMotionParam := (diAccInMS:=500,diDecInMS:=500,diAutoSpdInUMPS:=50000); (*covered 150, w/o cover 50*)
		tyLifterTuning : tyMotionCANTuning := (diAsdaA2Inertia:=62,diAsdaA2PosLoopGain:=64,diAsdaA2PosFFGain:=50,diAsdaA2SpdLoopGain:=257,diAsdaA2SpdIntegral:=41,diAsdaA2LowPassFltr:=40,diAsdaA2AntiInterGain:=41,diAsdaA2FirstTorqueCmd:=300,diLex28LTNDderivativeGain_P800:=1116,diLex28LTNIintegralGain_P801:=321,diLex28LTNIVdeIntlGain_P802:=319,diLex28LTNPpropotionalGain_P803:=482,diLex28LTNUSERGAIN_P804:=1000,diLex28NLAFFLPFHZspringFil_P805:=5000,diLex28NLFILTDAMPING_P814:=35,diLex28NLFILTT1_P815:=25,diPronetInertia:=0,diPronetRealTimeAutoAdjSet:=0,diPronetPosLoopGain:=40,diPronetSpdLoopGain:=250,diPronetSpdIntegral:=500,diPronetTorqueFilter:=100,diPronetPosFeedForward:=0,diPronetLowSpeedTestFiltering:=10,diPronetStopMode:=5);
		eLifterServoMotorType : eServoMotorType := DeltaAsdaA2; (*Selection of  Motor Brand*)
		sDIProgNm : STRING[15] := 'DInput';
		sAGVSvrProgNm : STRING[15] := 'AGVServer';
		sAGVMag1ProgNm : STRING[15] := 'AGVMag 1';
		sAGVMag2ProgNm : STRING[15] := 'AGVMag 2';
		sAGVMag3ProgNm : STRING[15] := 'AGVMag 3';
		sAGVMag4ProgNm : STRING[15] := 'AGVMag 4';
		sHermesProgNm : STRING[15] := 'Hermes';
		sHermesRetainFileNm : STRING[80] := 'Hermes.dat';
		sHermesConfigFileNm : STRING[80] := 'Hermes.dat';
		sDSHermesAProgNm : STRING[15] := 'DSHermes A';
		udiDSHermesAFileKeepDay : UDINT := 7;
		udiDSHermesAAliveTmInSec : UDINT := 5;
		tDSHermesAConnTO : TIME := T#30s;
		sDSHermesBProgNm : STRING[15] := 'DSHermes B';
		udiDSHermesBFileKeepDay : UDINT := 7;
		udiDSHermesBAliveTmInSec : UDINT := 5;
		tDSHermesBConnTO : TIME := T#30s;
		sRmtHermesProgNm : STRING[15] := 'RmtHermes';
		sRmtHermesConfigFileNm : STRING[80] := 'RmtHermes.dat';
		udiRmtHermesFileKeepDay : UDINT := 7;
		udiRmtHermesAliveTmInSec : UDINT := 5;
		udiRmtHermesSndBffrSize : UDINT := 65536;
		udiRmtHermesRcvBffrSize : UDINT := 65536;
		sLFLeaderProgNm : STRING[15] := 'LFLeader';
		tLFLeaderOnlineChkDlyTm : TIME := T#30s;
		tLFLeaderSetTmOffDlyTm : TIME := T#10s;
		sLFFollowerProgNm : STRING[15] := 'Follower';
		sFollower1ProgNm : STRING[15] := 'Follower 1';
		sFollower2ProgNm : STRING[15] := 'Follower 2';
		sLCSProgNm : STRING[15] := 'LCS';
		sLCSMngRcpProgNm : STRING[15] := 'LCSMngRcp';
		sLCSLFProgNm : STRING[15] := 'LCSLF';
		sOpsTravLifLDProgNm : STRING[15] := 'OpsTravLifLD';
		sOpsMagLD1ProgNm : STRING[15] := 'OpsMagLD 1';
		sOpsMagLD2ProgNm : STRING[15] := 'OpsMagLD 2';
		sOpsMagLD3ProgNm : STRING[15] := 'OpsMagLD 3';
		sOpsMagLD4ProgNm : STRING[15] := 'OpsMagLD 4';
		sOpsMagConvLD1ProgNm : STRING[15] := 'OpsMagConvLD 1';
		sOpsMagConvLD2ProgNm : STRING[15] := 'OpsMagConvLD 2';
		sOpsMagConvLD3ProgNm : STRING[15] := 'OpsMagConvLD 3';
		sOpsMagConvLD4ProgNm : STRING[15] := 'OpsMagConvLD 4';
		sOpsLifMagLDProgNm : STRING[15] := 'OpsLifMagLD';
		tyProdRcpWidth : tyUILmt := (diMax:=400000,diMin:=70000);
		tyProdRcpMinSlt : tyUILmt := (diMax:=60,diMin:=5);
		tyProdRcpMaxSlt : tyUILmt := (diMax:=60,diMin:=5);
		tyProdRcpPitch : tyUILmt := (diMax:=55,diMin:=1);
		tyProdRcpMcModA : tyUILmt := (diMax:=0,diMin:=0);
		tyProdRcpMcModAB : tyUILmt := (diMax:=2,diMin:=0);
		tyUISSaverTm : tyUILmt := (diMax:=1800,diMin:=10);
		tyUIConvInitTm : tyUILmt := (diMax:=60000,diMin:=3000);
		tyUIMagConvRunTm : tyUILmt := (diMax:=60000,diMin:=5000);
		tyUITranOutErrDlyTm : tyUILmt := (diMax:=120000,diMin:=5000);
		tyUIHermesSndAliveTm : tyUILmt := (diMax:=1800000,diMin:=5000);
		tyUIHermesLnID : tyUILmt := (diMax:=1000,diMin:=1);
		tyUIAntiGapSenOnTm : tyUILmt := (diMax:=5000,diMin:=0);
		tyUIAntiGapSenOffTm : tyUILmt := (diMax:=5000,diMin:=0);
		tyUISltToSltDist : tyUILmt := (diMax:=70000,diMin:=1000);
		tyUIAWTargetPos : tyUILmt := (diMax:=240000,diMin:=0);
		tyUIAWStepSize : tyUILmt := (diMax:=240000,diMin:=-240000);
		tyUIAWNomSpd : tyUILmt := (diMax:=15000,diMin:=5000);
		tyUIAWSlwSpd : tyUILmt := (diMax:=15000,diMin:=5000);
		tyUITravTargetPos : tyUILmt := (diMax:=1500000,diMin:=-20000);
		tyUITravStepSize : tyUILmt := (diMax:=1500000,diMin:=-1500000);
		tyUITravNomSpd : tyUILmt := (diMax:=100000,diMin:=5000);
		tyUITravSlwSpd : tyUILmt := (diMax:=100000,diMin:=5000);
		tyUILifterTargetPos : tyUILmt := (diMax:=550000,diMin:=-10000);
		tyUILifterStepSize : tyUILmt := (diMax:=550000,diMin:=-550000);
		tyUILifterNomSpd : tyUILmt := (diMax:=100000,diMin:=5000);
		tyUILifterSlwSpd : tyUILmt := (diMax:=100000,diMin:=5000);
		tyUILFIndexBeforeOven : tyUILmt := (diMax:=100,diMin:=1);
		tyUILFIndexAfterOven : tyUILmt := (diMax:=100,diMin:=1);
		sUIDefaultLoginNm : STRING[30] := 'admin';
		sUIDefaultLoginPw : STRING[30] := 'admin';
		sPullerProgNm : STRING[15] := 'Puller';
		bPullerTwoCtrlIn : BOOL := TRUE;
		tPullerExtTO : TIME := T#15s;
		tPullerRetTO : TIME := T#15s;
		bProjPullerRotCylPrep : BOOL := TRUE;
		diProjPullerExtMaxSlt : DINT := 60;
		diProjPullerExtMinSlt : DINT := 4;
		tShutterWaitTmr : TIME := T#500ms;
		tyUIAWOffset : tyUILmt := (diMax:=2000,diMin:=-2000);
		bMagAutoVerifyPrep : BOOL := FALSE;
		tyUIMcParamMagAutoEntSenTm : tyUILmt := (diMax:=5000,diMin:=0);
		bProjDBAOnRgtSen : BOOL := FALSE;
		bAutoLogoutPrep : BOOL := FALSE;
		tyUIAutoLogoutTm : tyUILmt := (diMax:=1800000,diMin:=60000);
		sMpNtParamFileNm : STRING[255] := 'NutekParameter.xml';
		sMpNtParamPVNm : STRING[100] := 'NtParam:tyMpNtParamCurr1';
		bLFProdWidth2Prep : BOOL := FALSE;
		tLFFollowerOnlineChkDlyTm : TIME := T#30s;
		tyNetworkMode : tyUILmt := (diMax:=1,diMin:=0);
		sUSSOT1ProgNm : STRING[15] := 'USSOT1';
		tUSSOT1RstDlyTm : TIME := T#0s;
		tUSSOT1SigInChkTm : TIME := T#100ms;
		sUSSOT2ProgNm : STRING[15] := 'USSOT2';
		tUSSOT2RstDlyTm : TIME := T#0s;
		tUSSOT2SigInChkTm : TIME := T#100ms;
		sUSSOT3ProgNm : STRING[15] := 'USSOT3';
		tUSSOT3RstDlyTm : TIME := T#0s;
		tUSSOT3SigInChkTm : TIME := T#100ms;
		sUSSOT4ProgNm : STRING[15] := 'USSOT4';
		tUSSOT4RstDlyTm : TIME := T#0s;
		tUSSOT4SigInChkTm : TIME := T#100ms;
		sDSSOT1ProgNm : STRING[15] := 'DSSOT1';
		tDSSOT1RstDlyTm : TIME := T#0s;
		tDSSOT1SigInChkTm : TIME := T#100ms;
		sDSSOT2ProgNm : STRING[15] := 'DSSOT2';
		tDSSOT2RstDlyTm : TIME := T#0s;
		tDSSOT2SigInChkTm : TIME := T#100ms;
		sDSSOT3ProgNm : STRING[15] := 'DSSOT3';
		tDSSOT3RstDlyTm : TIME := T#0s;
		tDSSOT3SigInChkTm : TIME := T#100ms;
		sDSSOT4ProgNm : STRING[15] := 'DSSOT4';
		tDSSOT4RstDlyTm : TIME := T#0s;
		tDSSOT4SigInChkTm : TIME := T#100ms;
		sMachineProgNm : STRING[15] := 'Machine';
		sMachine1ProgNm : STRING[15] := 'Machine1';
		sUSBRdrProgNm : STRING[15] := 'USBReader';
		bUSBScannerPrep : BOOL := FALSE;
		bBCodeScannerPrep : BOOL := FALSE;
		bScanPrep : BOOL := FALSE;
		tyVID : tyUILmt := (diMax:=65535,diMin:=0);
		tyPID : tyUILmt := (diMax:=65535,diMin:=0);
		bSOTReadyOnFirst : BOOL := TRUE;
		bShowMESName : BOOL := FALSE;
		bShowFMorMESActive : BOOL := FALSE;
		eScannerType : eScannerType := RS232;
		bRS232ScannerPrep : BOOL := FALSE;
		sRS232ProgNm : STRING[15] := 'RS232';
		tyProdRcpMtrPshrExtSpd : tyUILmt := (diMax:=8,diMin:=1);
		tyProdRcpMtrPshrExtTorq : tyUILmt := (diMax:=100,diMin:=10);
		diPullerHeightInMM : DINT := 54;
		bProjDSFixToFixRail : BOOL := FALSE;
		bProjWorkOrderOPCUA : BOOL := FALSE;
		bProjServoPullerPusherPrep : BOOL := FALSE;
		sPPProgNm : STRING[15] := 'ServoPullPusher';
		sPPDevice : STRING[3] := 'IF7';
		usiPPNode : USINT := 20;
		bPPDir : BOOL := FALSE;
		bPPDirBl : BOOL := FALSE;
		diPPPitchInUM : DINT := 3000; (*NA*)
		diPPMovBlDistInUM : DINT := 0;
		tyPPParamInHm : tyMotionCANParamInHm := (diStartVelInUMPS:=15000,diAcc:=25);
		tyPPParamInConvert : tyMotionCANParamInConvert := (diPitchInUM:=3000); (*estun1048576*)
		tyPPParam : tyMotionParam := (diAccInMS:=500,diDecInMS:=500,diAutoSpdInUMPS:=150000);
		tyPPTuning : tyMotionCANTuning := (diAsdaA2Inertia:=76,diAsdaA2PosLoopGain:=53,diAsdaA2PosFFGain:=50,diAsdaA2SpdLoopGain:=213,diAsdaA2SpdIntegral:=34,diAsdaA2LowPassFltr:=49,diAsdaA2AntiInterGain:=34,diAsdaA2FirstTorqueCmd:=300,diLex28LTNDderivativeGain_P800:=0,diLex28LTNIintegralGain_P801:=0,diLex28LTNIVdeIntlGain_P802:=0,diLex28LTNPpropotionalGain_P803:=0,diLex28LTNUSERGAIN_P804:=0,diLex28NLAFFLPFHZspringFil_P805:=0,diLex28NLFILTDAMPING_P814:=0,diLex28NLFILTT1_P815:=0,diPronetInertia:=0,diPronetRealTimeAutoAdjSet:=0,diPronetPosLoopGain:=80,diPronetSpdLoopGain:=750,diPronetSpdIntegral:=600,diPronetTorqueFilter:=4,diPronetPosFeedForward:=0,diPronetLowSpeedTestFiltering:=0,diPronetStopMode:=5);
		ePPServoMotorType : eServoMotorType := DeltaAsdaA2; (*Selection of  Motor Brand*)
		bProjCurtainSenPrep : BOOL := FALSE; (*Shutter Keep Ret(Open)*)
		bProjMagHeightChkPrep : BOOL := FALSE;
		diTravGoToMagWidthChkPt1 : DINT := 3000;
		diTravGoToMagWidthChkPt2 : DINT := 3000;
		diTravGoToMagWidthChkPt3 : DINT := 3000;
		tyPPTorqParam : PPTorqParam := (usiStartTorque:=22,uiRatio:=889); (*Ratio= x/100*)
		bProjLifTravMnlLoad : BOOL := FALSE;
		eCustomerReq : eCustomer := NA;
		bProjShutter2Prep : BOOL := FALSE;
		bProjShutter3Prep : BOOL := FALSE;
		bHermesSvyPrep : BOOL := FALSE; (*Supervisory Hermes Preparation*)
		bHermesSvyFirstMcInTheLine : BOOL := FALSE; (*Turn On this for Loader / Destacker Only. Other type of machine turns off.*)
		bHermesSvyMagTypeMc : BOOL := FALSE; (*Turn On this for Loader (Magazine type machine) Only. Other type of machine turns off.
*)
		sSvyHermesProgNm : STRING[15] := 'SvyHermes';
		sSvyHermesConfigFileNm : STRING[80] := 'SvyHermes.dat';
		udiSvyHermesFileKeepDay : UDINT := 7;
		udiSvyHermesAliveTmInSec : UDINT := 5;
		tSvyHermesConnTO : TIME := T#30s;
		sSvyHermesRetainFileNm : STRING[80] := 'WorkOrder.dat';
		sDSHermesRetainFileNm : STRING[80] := 'BoardData.dat';
		rMachineCycleTime : REAL := 6.0; (*1.0 = 1 second*)
		rAutoWidthCycleTime : REAL := 30.0; (*30.0 = 30 seconds*)
		bHermesScannerPrep : BOOL := FALSE; (*Turn On if machine has fixed scanner or handheld scanner*)
		iInput : INT := 1; (*Total Inlet, Single Track = 1, Dual Track = 2, and so on*)
		iOutput : INT := 1; (*Total Outlet, Single Track = 1, Dual Track = 2, and so on*)
		bProjAutoRcpPrep : BOOL := FALSE;
		tyAutoRcpParamLmt : AutoRcpLmt := (diThicknessInUM:=5500,diMaxTopClearamceInUM:=30000,diMaxBottomCleranceInUM:=6700);
		eAutoRcpPrecededBy : eAutoRcpPreceded := PrecededBySelf;
		bchineseprep : BOOL := FALSE;
		bgermanprep : BOOL := FALSE;
		bProjOutShutter2Prep : BOOL := FALSE;
		siProjCntrPullLmt : SINT := -1; (*(-1) index to next slot ; (x) no. of brd to alarm*)
		bUIConvDirRL : BOOL := FALSE;
		bProjTrolleyLckPrep : BOOL := FALSE;
		sTrolleyLckProgNm : STRING[15] := 'TrolleyLck';
		bTrolleyLckTwoCtrlIn : BOOL := FALSE;
		tTrolleyLckExtTO : TIME := T#6s;
		tTrolleyLckRetTO : TIME := T#6s;
		sTrolleyLckProgNm2 : STRING[15] := 'TrolleyLck2';
		bTrolleyLckTwoCtrlIn2 : BOOL := FALSE;
		tTrolleyLckExtTO2 : TIME := T#6s;
		tTrolleyLckRetTO2 : TIME := T#6s;
	END_STRUCT;
END_TYPE

(**)

TYPE
	tyUILmt : 	STRUCT
		diMax : DINT;
		diMin : DINT;
	END_STRUCT;
	PPTorqParam : 	STRUCT
		usiStartTorque : USINT;
		uiRatio : UINT;
	END_STRUCT;
	eScannerType :
		(
		RS232,
		USB
		);
	eCustomer :
		(
		NA,
		Bosch_China,
		Bosch_Portugal,
		Bosch_America,
		Bosch_Malaysia,
		Siemens,
		We_Fabricate,
		reserve1,
		reserve2,
		reserve3,
		reserve4,
		reserve5,
		reserve6,
		reserve7,
		reserve8,
		reserve9
		);
END_TYPE

(**)
(*Auto Rcp*)

TYPE
	eAutoRcpPreceded :
		(
		PrecededBySelf,
		PrecededByF1,
		PrecededByF2
		);
	AutoRcpLmt : 	STRUCT
		diThicknessInUM : DINT;
		diMaxTopClearamceInUM : DINT;
		diMaxBottomCleranceInUM : DINT;
		reserve1 : DINT;
		reserve2 : DINT;
		reserve3 : DINT;
	END_STRUCT;
END_TYPE
```

### NtParam.var
```iecst
(*2019-05-20*)
(**)
(*Action & State & Status*)
VAR
	p_NtParamStat : UDINT;
	p_NtParamStatus : UDINT;
	p_NtParamStatTxt : UDINT;
END_VAR
(**)
(*Alarm*)
VAR
	p_NtParamAlmData : UDINT;
END_VAR
(**)
(*Output*)
VAR
	p_NtParamFileNotFound : UDINT;
END_VAR
(**)
VAR
	p_NtParamCurr : UDINT;
END_VAR
(**)
VAR
	p_NtParamDISettings : UDINT;
	p_NtParamDOSettings : UDINT;
	p_NtParamAWPusherPrep : UDINT;
	p_NtParamAWPrep : UDINT;
	p_NtParamLFPrep : UDINT;
	p_NtParamLeaderMc : UDINT;
	p_NtParamLFUsrSetPrep : UDINT;
	p_NtParamLFWidthLimit : UDINT;
	p_NtParamLFProdWidthChk : UDINT;
	p_NtParamDSWidthChkPrep : UDINT;
	p_NtParamLCSLFPrep : UDINT;
	p_NtParamLCSReqRcpPrep : UDINT;
	p_NtParamLCSManageRcpPrep : UDINT;
	p_NtParamLCSLiveDatPrep : UDINT;
	p_NtParamIPCSMEMA9851ExtdPrep : UDINT;
	p_NtParamVSMEMAPrep : UDINT;
	p_NtParamHermesPrep : UDINT;
	p_NtParamHermesRmtPrep : UDINT;
	p_NtParamSSaverPrep : UDINT;
	p_NtParamPushPulAWidthOffset : UDINT;
	p_NtParamWidthOffset : UDINT;
	p_NtParamJobNo : UDINT;
	p_NtParamNtAddr : UDINT;
	p_NtParamShutterWaitTmr : UDINT;
END_VAR
(**)
VAR
	p_NtParamProjLaneBPrep : UDINT;
	p_NtParamProjTopToBtmDefault : UDINT;
	p_NtParamProjLongBrdPrep : UDINT;
	p_NtParamProjInletShutPrep : UDINT;
	p_NtParamProjOutletShutPrep : UDINT;
	p_NtParamProjMag1ConvPrep : UDINT;
	p_NtParamProjMag2ConvPrep : UDINT;
	p_NtParamProjMag3ConvPrep : UDINT;
	p_NtParamProjMag4ConvPrep : UDINT;
	p_NtParamProjMagOrientChkSenPrep : UDINT;
	p_NtParamProjAGVPrep : UDINT;
	p_NtParamProjAGVInPosSenPrep : UDINT;
	p_NtParamProjBypsInitConvPrep : UDINT;
	p_NtParamProjRlsNewProdPrep : UDINT;
	p_NtParamProjBtnInsertRmvMag : UDINT;
	p_NtParamProjMagMinSlt : UDINT;
	p_NtParamProjMagMaxSlt : UDINT;
	p_NtParamProjMag : UDINT;
	p_NtParamProjConvDir : UDINT;
	p_NtParamProjMagConvDir : UDINT;
	p_NtParamProjMagAutoVerifyPrep : UDINT;
	p_NtParamProjMotorizedPullerPrep : UDINT;
	p_NtParamProjMagSafetyBarPrep : UDINT;
	p_NtParamProjLifterMagPlatform : UDINT;
END_VAR
(**)
VAR
	p_NtParamUsrFolderProgNm : UDINT;
END_VAR
(**)
VAR
	p_NtParamLibVersionProgNm : UDINT;
END_VAR
(**)
VAR
	p_NtParamTimeProgNm : UDINT;
END_VAR
(**)
VAR
	p_NtParamHWInfoProgNm : UDINT;
	p_NtParamHWInfoDevice : UDINT;
END_VAR
(**)
(*TLBuz*)
VAR
	p_NtParamTLBuzMode : UDINT;
	p_NtParamTLChgRcpBlinkTm : UDINT;
END_VAR
(**)
VAR
	p_NtParamTLErrBlinkTm : UDINT;
	p_NtParamBuzErrOnTm : UDINT;
	p_NtParamBuzErrRestTm : UDINT;
	p_NtParamBuzErrOnCntr : UDINT;
	p_NtParamBuzErrStopSeqEn : UDINT;
	p_NtParamBuzErrStopSeqCntr : UDINT;
END_VAR
(**)
VAR
	p_NtParamTLWarnBlinkTm : UDINT;
	p_NtParamBuzWarnOnTm : UDINT;
	p_NtParamBuzWarnRestTm : UDINT;
	p_NtParamBuzWarnOnCntr : UDINT;
	p_NtParamBuzWarnStopSeqEn : UDINT;
	p_NtParamBuzWarnStopSeqCntr : UDINT;
END_VAR
(**)
VAR
	p_NtParamTLWarn1BlinkTm : UDINT;
	p_NtParamBuzWarn1OnTm : UDINT;
	p_NtParamBuzWarn1RestTm : UDINT;
	p_NtParamBuzWarn1OnCntr : UDINT;
	p_NtParamBuzWarn1StopSeqEn : UDINT;
	p_NtParamBuzWarn1StopSeqCntr : UDINT;
END_VAR
(**)
VAR
	p_NtParamTLWarn2BlinkTm : UDINT;
	p_NtParamBuzWarn2OnTm : UDINT;
	p_NtParamBuzWarn2RestTm : UDINT;
	p_NtParamBuzWarn2OnCntr : UDINT;
	p_NtParamBuzWarn2StopSeqEn : UDINT;
	p_NtParamBuzWarn2StopSeqCntr : UDINT;
END_VAR
(**)
VAR
	p_NtParamTLWarn3BlinkTm : UDINT;
	p_NtParamBuzWarn3OnTm : UDINT;
	p_NtParamBuzWarn3RestTm : UDINT;
	p_NtParamBuzWarn3OnCntr : UDINT;
	p_NtParamBuzWarn3StopSeqEn : UDINT;
	p_NtParamBuzWarn3StopSeqCntr : UDINT;
END_VAR
(**)
VAR
	p_NtParamTLWarn4BlinkTm : UDINT;
	p_NtParamBuzWarn4OnTm : UDINT;
	p_NtParamBuzWarn4RestTm : UDINT;
	p_NtParamBuzWarn4OnCntr : UDINT;
	p_NtParamBuzWarn4StopSeqEn : UDINT;
	p_NtParamBuzWarn4StopSeqCntr : UDINT;
END_VAR
(**)
VAR
	p_NtParamTLWarn5BlinkTm : UDINT;
	p_NtParamBuzWarn5OnTm : UDINT;
	p_NtParamBuzWarn5RestTm : UDINT;
	p_NtParamBuzWarn5OnCntr : UDINT;
	p_NtParamBuzWarn5StopSeqEn : UDINT;
	p_NtParamBuzWarn5StopSeqCntr : UDINT;
END_VAR
(**)
VAR
	p_NtParamBuzAlertOnTm : UDINT;
	p_NtParamBuzAlertRestTm : UDINT;
	p_NtParamBuzAlertOnCntr : UDINT;
	p_NtParamBuzAlertStopSeqEn : UDINT;
	p_NtParamBuzAlertStopSeqCntr : UDINT;
END_VAR
(**)
VAR
	p_NtParamTLBlueBlinkTm : UDINT;
	p_NtParamTLAmberBlinkTm : UDINT;
	p_NtParamTLWhiteBlinkTm : UDINT;
	p_NtParamTLRedBlinkTm : UDINT;
	p_NtParamTLGreenBlinkTm : UDINT;
END_VAR
(**)
VAR
	p_NtParamAlmProgNm : UDINT;
	p_NtParamAlmFileKeepDay : UDINT;
END_VAR
(**)
VAR
	p_NtParamProdRcpProgNm : UDINT;
	p_NtParamProdRcpListFileNm : UDINT;
	p_NtParamProdRcpSingleFileNm : UDINT;
END_VAR
(**)
VAR
	p_NtParamMpProdRcpProgNm : UDINT;
	p_NtParamMpProdRcpFileNm : UDINT;
	p_NtParamMpProdRcpPVNm : UDINT;
END_VAR
(**)
VAR
	p_NtParamMagRcpProgNm : UDINT;
	p_NtParamMagRcpListFileNm : UDINT;
	p_NtParamMagRcpSingleFileNm : UDINT;
END_VAR
(**)
VAR
	p_NtParamMagRcpProgNm1 : UDINT;
	p_NtParamMagRcpListFileNm1 : UDINT;
	p_NtParamMagRcpSingleFileNm1 : UDINT;
END_VAR
(**)
VAR
	p_NtParamMcParamProgNm : UDINT;
	p_NtParamMcParamFileNm : UDINT;
END_VAR
(**)
VAR
	p_NtParamUsrMgmtProgNm : UDINT;
END_VAR
(**)
VAR
	p_NtParamBffr1ProgNm : UDINT;
	p_NtParamBffr1FileNm : UDINT;
	p_NtParamBffr1FIFO : UDINT;
END_VAR
(**)
VAR
	p_NtParamBffr2ProgNm : UDINT;
	p_NtParamBffr2FileNm : UDINT;
	p_NtParamBffr2FIFO : UDINT;
END_VAR
(**)
VAR
	p_NtParamBffr3ProgNm : UDINT;
	p_NtParamBffr3FileNm : UDINT;
	p_NtParamBffr3FIFO : UDINT;
END_VAR
(**)
VAR
	p_NtParamBffr4ProgNm : UDINT;
	p_NtParamBffr4FileNm : UDINT;
	p_NtParamBffr4FIFO : UDINT;
END_VAR
(**)
VAR
	p_NtParamUSSMEMA1ProgNm : UDINT;
	p_NtParamUSSMEMA1RstDlyTm : UDINT;
	p_NtParamUSSMEMA1SigInChkTm : UDINT;
END_VAR
(**)
VAR
	p_NtParamUSSMEMA2ProgNm : UDINT;
	p_NtParamUSSMEMA2RstDlyTm : UDINT;
	p_NtParamUSSMEMA2SigInChkTm : UDINT;
END_VAR
(**)
VAR
	p_NtParamUSSMEMA3ProgNm : UDINT;
	p_NtParamUSSMEMA3RstDlyTm : UDINT;
	p_NtParamUSSMEMA3SigInChkTm : UDINT;
END_VAR
(**)
VAR
	p_NtParamUSSMEMA4ProgNm : UDINT;
	p_NtParamUSSMEMA4RstDlyTm : UDINT;
	p_NtParamUSSMEMA4SigInChkTm : UDINT;
END_VAR
(**)
VAR
	p_NtParamDSSMEMA1ProgNm : UDINT;
	p_NtParamDSSMEMA1RstDlyTm : UDINT;
	p_NtParamDSSMEMA1SigInChkTm : UDINT;
END_VAR
(**)
VAR
	p_NtParamDSSMEMA2ProgNm : UDINT;
	p_NtParamDSSMEMA2RstDlyTm : UDINT;
	p_NtParamDSSMEMA2SigInChkTm : UDINT;
END_VAR
(**)
VAR
	p_NtParamDSSMEMA3ProgNm : UDINT;
	p_NtParamDSSMEMA3RstDlyTm : UDINT;
	p_NtParamDSSMEMA3SigInChkTm : UDINT;
END_VAR
(**)
VAR
	p_NtParamDSSMEMA4ProgNm : UDINT;
	p_NtParamDSSMEMA4RstDlyTm : UDINT;
	p_NtParamDSSMEMA4SigInChkTm : UDINT;
END_VAR
(**)
VAR
	p_NtParamDSSMEMAAProgNm : UDINT;
	p_NtParamDSSMEMAARstDlyTm : UDINT;
	p_NtParamDSSMEMAASigInChkTm : UDINT;
END_VAR
(**)
VAR
	p_NtParamDSSMEMABProgNm : UDINT;
	p_NtParamDSSMEMABRstDlyTm : UDINT;
	p_NtParamDSSMEMABSigInChkTm : UDINT;
END_VAR
(**)
VAR
	p_NtParamInShutterProgNm : UDINT;
	p_NtParamInShutterTwoCtrlIn : UDINT;
	p_NtParamInShutterExtTO : UDINT;
	p_NtParamInShutterRetTO : UDINT;
END_VAR
(**)
VAR
	p_NtParamOutShutterProgNm : UDINT;
	p_NtParamOutShutterTwoCtrlIn : UDINT;
	p_NtParamOutShutterExtTO : UDINT;
	p_NtParamOutShutterRetTO : UDINT;
END_VAR
(**)
VAR
	p_NtParamSelClamp1ProgNm : UDINT;
	p_NtParamSelClamp1TwoCtrlIn : UDINT;
	p_NtParamSelClamp1ExtDlyTm : UDINT;
	p_NtParamSelClamp1RetDlyTm : UDINT;
END_VAR
(**)
VAR
	p_NtParamSelClamp2ProgNm : UDINT;
	p_NtParamSelClamp2TwoCtrlIn : UDINT;
	p_NtParamSelClamp2ExtDlyTm : UDINT;
	p_NtParamSelClamp2RetDlyTm : UDINT;
END_VAR
(**)
VAR
	p_NtParamSelClamp3ProgNm : UDINT;
	p_NtParamSelClamp3TwoCtrlIn : UDINT;
	p_NtParamSelClamp3ExtDlyTm : UDINT;
	p_NtParamSelClamp3RetDlyTm : UDINT;
END_VAR
(**)
VAR
	p_NtParamSelClamp4ProgNm : UDINT;
	p_NtParamSelClamp4TwoCtrlIn : UDINT;
	p_NtParamSelClamp4ExtDlyTm : UDINT;
	p_NtParamSelClamp4RetDlyTm : UDINT;
END_VAR
(**)
VAR
	p_NtParamPullConvProgNm : UDINT;
	p_NtParamPullConvOnDirMod : UDINT;
	p_NtParamPullConvMtrOffDlyTm : UDINT;
	p_NtParamPullConvPullExtTO : UDINT;
	p_NtParamPullConvPullRetTO : UDINT;
	p_NtParamPullConvRotHomeTO : UDINT;
	p_NtParamPullConvRotRemoteTO : UDINT;
END_VAR
(**)
VAR
	p_NtParamMagConv1ProgNm : UDINT;
	p_NtParamMagConv1OnDirMod : UDINT;
	p_NtParamMagConv1MtrOffDlyTm : UDINT;
	p_NtParamMagConv1ClprClampTO : UDINT;
	p_NtParamMagConv1ClprUnclampTO : UDINT;
END_VAR
(**)
VAR
	p_NtParamMagConv2ProgNm : UDINT;
	p_NtParamMagConv2OnDirMod : UDINT;
	p_NtParamMagConv2MtrOffDlyTm : UDINT;
	p_NtParamMagConv2ClprClampTO : UDINT;
	p_NtParamMagConv2ClprUnclampTO : UDINT;
END_VAR
(**)
VAR
	p_NtParamMagConv3ProgNm : UDINT;
	p_NtParamMagConv3OnDirMod : UDINT;
	p_NtParamMagConv3MtrOffDlyTm : UDINT;
	p_NtParamMagConv3ClprClampTO : UDINT;
	p_NtParamMagConv3ClprUnclampTO : UDINT;
END_VAR
(**)
VAR
	p_NtParamMagConv4ProgNm : UDINT;
	p_NtParamMagConv4OnDirMod : UDINT;
	p_NtParamMagConv4MtrOffDlyTm : UDINT;
	p_NtParamMagConv4ClprClampTO : UDINT;
	p_NtParamMagConv4ClprUnclampTO : UDINT;
END_VAR
(**)
VAR
	p_NtParamMtrPshrProgNm : UDINT;
	p_NtParamMtrPshrDir : UDINT;
	p_NtParamMtrPshrAlmRstTm : UDINT;
	p_NtParamMtrPshrAlmTrigTm : UDINT;
	p_NtParamMtrPshrExtTO : UDINT;
	p_NtParamMtrPshrRetTO : UDINT;
	p_NtParamMtrPshrExtSlowSpd : UDINT;
	p_NtParamMtrPshrRetSlowSpd : UDINT;
	p_NtParamMtrPshrExtNomSpd : UDINT;
	p_NtParamMtrPshrRetNomSpd : UDINT;
	p_NtParamMtrPshrExtTorq : UDINT;
	p_NtParamMtrPshrRetTorq : UDINT;
	p_NtParamMtrPshrStartTorq : UDINT;
END_VAR
(**)
VAR
	p_NtParamAWPushPulProgNm : UDINT;
	p_NtParamAWPushPulDevice : UDINT;
	p_NtParamAWPushPulNode : UDINT;
	p_NtParamAWPushPulDir : UDINT;
	p_NtParamAWPushPulDirBl : UDINT;
	p_NtParamAWPushPulPitchInUM : UDINT;
	p_NtParamAWPushPulMovBlDistInUM : UDINT;
	p_NtParamAWPushPulParamInHm : UDINT;
	p_NtParamAWPushPulParamInConvert : UDINT;
	p_NtParamAWPushPulParam : UDINT;
	p_NtParamAWPushPulAcc : UDINT;
	p_NtParamAWPushPulDec : UDINT;
	p_NtParamAWPushPulAutoSpd : UDINT;
	p_NtParamAWPushPulTuning : UDINT;
	p_NtParamAWPushPulMotorType : UDINT;
END_VAR
(**)
VAR
	p_NtParamAWProgNm : UDINT;
	p_NtParamAWDevice : UDINT;
	p_NtParamAWNode : UDINT;
	p_NtParamAWDir : UDINT;
	p_NtParamAWDirBl : UDINT;
	p_NtParamAWPitchInUM : UDINT;
	p_NtParamAWMovBlDistInUM : UDINT;
	p_NtParamAWParamInHm : UDINT;
	p_NtParamAWParamInConvert : UDINT;
	p_NtParamAWParam : UDINT;
	p_NtParamAWAcc : UDINT;
	p_NtParamAWDec : UDINT;
	p_NtParamAWAutoSpd : UDINT;
	p_NtParamAWTuning : UDINT;
	p_NtParamAWMotorType : UDINT;
END_VAR
(**)
VAR
	p_NtParamTravProgNm : UDINT;
	p_NtParamTravDevice : UDINT;
	p_NtParamTravNode : UDINT;
	p_NtParamTravDir : UDINT;
	p_NtParamTravParamInHm : UDINT;
	p_NtParamTravParamInConvert : UDINT;
	p_NtParamTravParam : UDINT;
	p_NtParamTravAcc : UDINT;
	p_NtParamTravDec : UDINT;
	p_NtParamTravAutoSpd : UDINT;
	p_NtParamTravTuning : UDINT;
	p_NtParamTravMotorType : UDINT;
	p_NtParamTravLongBrdAutoSpd : UDINT;
END_VAR
(**)
VAR
	p_NtParamLifterProgNm : UDINT;
	p_NtParamLifterDevice : UDINT;
	p_NtParamLifterNode : UDINT;
	p_NtParamLifterDir : UDINT;
	p_NtParamLifterParamInHm : UDINT;
	p_NtParamLifterParamInConvert : UDINT;
	p_NtParamLifterParam : UDINT;
	p_NtParamLifterAcc : UDINT;
	p_NtParamLifterDec : UDINT;
	p_NtParamLifterAutoSpd : UDINT;
	p_NtParamLifterMotorType : UDINT;
	p_NtParamLifterTuning : UDINT;
END_VAR
(**)
VAR
	p_NtParamDIProgNm : UDINT;
END_VAR
(**)
VAR
	p_NtParamAIVSvrProgNm : UDINT;
END_VAR
(**)
VAR
	p_NtParamAGVMag1ProgNm : UDINT;
	p_NtParamAGVMag2ProgNm : UDINT;
	p_NtParamAGVMag3ProgNm : UDINT;
	p_NtParamAGVMag4ProgNm : UDINT;
END_VAR
(**)
VAR
	p_NtParamHermesProgNm : UDINT;
	p_NtParamHermesRetainFileNm : UDINT;
	p_NtParamHermesConfigFileNm : UDINT;
END_VAR
(**)
VAR
	p_NtParamDSHermesAProgNm : UDINT;
	p_NtParamDSHermesAFileKeepDay : UDINT;
	p_NtParamDSHermesAAliveTmInSec : UDINT;
	p_NtParamDSHermesAConnTO : UDINT;
END_VAR
(**)
VAR
	p_NtParamDSHermesBProgNm : UDINT;
	p_NtParamDSHermesBFileKeepDay : UDINT;
	p_NtParamDSHermesBAliveTmInSec : UDINT;
	p_NtParamDSHermesBConnTO : UDINT;
END_VAR
(**)
VAR
	p_NtParamRmtHermesProgNm : UDINT;
	p_NtParamRmtHermesConfigFileNm : UDINT;
	p_NtParamRmtHermesFileKeepDay : UDINT;
	p_NtParamRmtHermesAliveTmInSec : UDINT;
	p_NtParamRmtHermesSndBffrSize : UDINT;
	p_NtParamRmtHermesRcvBffrSize : UDINT;
END_VAR
(**)
VAR
	p_NtParamHermesSvyPrep : UDINT;
	p_NtParamHermesSvyFirstMc : UDINT;
	p_NtParamHermesSvyMagTypeMc : UDINT;
	p_NtParamSvyHermesProgNm : UDINT;
	p_NtParamSvyHermesConfigFileNm : UDINT;
	p_NtParamSvyHermesFileKeepDay : UDINT;
	p_NtParamSvyHermesAliveTmInSec : UDINT;
	p_NtParamSvyHermesConnTO : UDINT;
	p_NtParamSvyHermesRetainFileNm : UDINT;
	p_NtParamDSHermesRetainFileNm : UDINT;
	p_NtParamDSHermesMcCycleTm : UDINT;
	p_NtParamDSHermesAWCycleTm : UDINT;
	p_NtParamHermesScannerPrep : UDINT;
	p_NtParamHermesInput : UDINT;
	p_NtParamHermesOutput : UDINT;
END_VAR
(**)
VAR
	p_NtParamLFLeaderProgNm : UDINT;
	p_NtParamLFLeaderOnlineChkDlyTm : UDINT;
	p_NtParamLFLeaderSetTmOffDlyTm : UDINT;
END_VAR
(**)
VAR
	p_NtParamLFFollowerProgNm : UDINT;
END_VAR
(**)
VAR
	p_NtParamFollower1ProgNm : UDINT;
	p_NtParamFollower2ProgNm : UDINT;
END_VAR
(**)
VAR
	p_NtParamLCSProgNm : UDINT;
END_VAR
(**)
VAR
	p_NtParamLCSMngRcpProgNm : UDINT;
END_VAR
(**)
VAR
	p_NtParamLCSLFProgNm : UDINT;
END_VAR
(**)
VAR
	p_NtParamOpsTravLifLDProgNm : UDINT;
END_VAR
(**)
VAR
	p_NtParamOpsMagLD1ProgNm : UDINT;
END_VAR
(**)
VAR
	p_NtParamOpsMagLD2ProgNm : UDINT;
END_VAR
(**)
VAR
	p_NtParamOpsMagLD3ProgNm : UDINT;
END_VAR
(**)
VAR
	p_NtParamOpsMagLD4ProgNm : UDINT;
END_VAR
(**)
VAR
	p_NtParamOpsMagConvLD1ProgNm : UDINT;
END_VAR
(**)
VAR
	p_NtParamOpsMagConvLD2ProgNm : UDINT;
END_VAR
(**)
VAR
	p_NtParamOpsMagConvLD3ProgNm : UDINT;
END_VAR
(**)
VAR
	p_NtParamOpsMagConvLD4ProgNm : UDINT;
END_VAR
(**)
VAR
	p_NtParamOpsLifMagLDProgNm : UDINT;
END_VAR
(**)
VAR
	p_NtParamProdRcpMinWidth : UDINT;
	p_NtParamProdRcpMaxWidth : UDINT;
	p_NtParamProdRcpMinMinSlt : UDINT;
	p_NtParamProdRcpMaxMinSlt : UDINT;
	p_NtParamProdRcpMinMaxSlt : UDINT;
	p_NtParamProdRcpMaxMaxSlt : UDINT;
	p_NtParamProdRcpMinPitch : UDINT;
	p_NtParamProdRcpMaxPitch : UDINT;
	p_NtParamProdRcpMinMcModA : UDINT;
	p_NtParamProdRcpMaxMcModA : UDINT;
	p_NtParamProdRcpMinMcModAB : UDINT;
	p_NtParamProdRcpMaxMcModAB : UDINT;
END_VAR
(**)
VAR
	p_NtParamPullerProgNm : UDINT;
	p_NtParamPullerTwoCtrlIn : UDINT;
	p_NtParamPullerExtTO : UDINT;
	p_NtParamPullerRetTO : UDINT;
	p_NtParamProjPullerRotCylPrep : UDINT;
	p_NtParamProjPullerExtMaxSlt : UDINT;
	p_NtParamProjPullerExtMinSlt : UDINT;
END_VAR
(**)
VAR
	p_NtParamProjDBAOnRgtSen : UDINT;
	p_NtParamLFWidth2Prep : UDINT;
	p_NtParamLFFllowerOnlineChkDlyTm : UDINT;
END_VAR
(**)
VAR
	p_NtParamUSSOT1ProgNm : UDINT;
	p_NtParamUSSOT1RstDlyTm : UDINT;
	p_NtParamUSSOT1SigInChkTm : UDINT;
	p_NtParamUSSOT2ProgNm : UDINT;
	p_NtParamUSSOT2RstDlyTm : UDINT;
	p_NtParamUSSOT2SigInChkTm : UDINT;
	p_NtParamUSSOT3ProgNm : UDINT;
	p_NtParamUSSOT3RstDlyTm : UDINT;
	p_NtParamUSSOT3SigInChkTm : UDINT;
	p_NtParamUSSOT4ProgNm : UDINT;
	p_NtParamUSSOT4RstDlyTm : UDINT;
	p_NtParamUSSOT4SigInChkTm : UDINT;
END_VAR
(**)
VAR
	p_NtParamDSSOT1ProgNm : UDINT;
	p_NtParamDSSOT1RstDlyTm : UDINT;
	p_NtParamDSSOT1SigInChkTm : UDINT;
	p_NtParamDSSOT2ProgNm : UDINT;
	p_NtParamDSSOT2RstDlyTm : UDINT;
	p_NtParamDSSOT2SigInChkTm : UDINT;
	p_NtParamDSSOT3ProgNm : UDINT;
	p_NtParamDSSOT3RstDlyTm : UDINT;
	p_NtParamDSSOT3SigInChkTm : UDINT;
	p_NtParamDSSOT4ProgNm : UDINT;
	p_NtParamDSSOT4RstDlyTm : UDINT;
	p_NtParamDSSOT4SigInChkTm : UDINT;
END_VAR
(**)
VAR
	p_NtParamProjSOTSenPrep : UDINT;
	p_NtParamMcProgNm : UDINT;
	p_NtParamMc1ProgNm : UDINT;
	p_NtParamProjUSBPrep : UDINT;
	p_NtParamUSBProgNm : UDINT;
	p_NtParamSOTReadyOnFirst : UDINT;
	p_NtParamShowMESName : UDINT;
	p_NtParamShowFMorMESActive : UDINT;
	p_NtParamRS232Prep : UDINT;
	p_NtParamRS232ProgNm : UDINT;
END_VAR
(**)
VAR
	p_NtParamProdRcpMinMtrPshrExtSpd : UDINT;
	p_NtParamProdRcpMaxMtrPshrExtSpd : UDINT;
	p_NtParamProdRcpMinMtrPshrExtToq : UDINT;
	p_NtParamProdRcpMaxMtrPshrExtToq : UDINT;
END_VAR
(**)
VAR
	p_NtParamMag1SafetyBarProgNm : UDINT;
	p_NtParamMag1SafetyBarTwoCtrlIn : UDINT;
	p_NtParamMag1SafetyBarExtTO : UDINT;
	p_NtParamMag1SafetyBarRetTO : UDINT;
END_VAR
(**)
VAR
	p_NtParamMag2SafetyBarProgNm : UDINT;
	p_NtParamMag2SafetyBarTwoCtrlIn : UDINT;
	p_NtParamMag2SafetyBarExtTO : UDINT;
	p_NtParamMag2SafetyBarRetTO : UDINT;
END_VAR
(**)
VAR
	p_NtParamMag3SafetyBarProgNm : UDINT;
	p_NtParamMag3SafetyBarTwoCtrlIn : UDINT;
	p_NtParamMag3SafetyBarExtTO : UDINT;
	p_NtParamMag3SafetyBarRetTO : UDINT;
END_VAR
(**)
VAR
	p_NtParamMag4SafetyBarProgNm : UDINT;
	p_NtParamMag4SafetyBarTwoCtrlIn : UDINT;
	p_NtParamMag4SafetyBarExtTO : UDINT;
	p_NtParamMag4SafetyBarRetTO : UDINT;
END_VAR
(**)
VAR
	p_NtParamPullerHeightInMM : UDINT;
	p_NtParamProjDsFixToFixRail : UDINT;
	p_NtParamProjWorkOrderOPCUA : UDINT;
END_VAR
(**)
VAR
	p_NtParamProjServoPullPusherPrep : UDINT;
	p_NtParamPPProgNm : UDINT;
	p_NtParamPPDevice : UDINT;
	p_NtParamPPNode : UDINT;
	p_NtParamPPDir : UDINT;
	p_NtParamPPDirBl : UDINT;
	p_NtParamPPPitchInUM : UDINT;
	p_NtParamPPMovBlDistInUM : UDINT;
	p_NtParamPPParamInHm : UDINT;
	p_NtParamPPParamInConvert : UDINT;
	p_NtParamPPParam : UDINT;
	p_NtParamPPAcc : UDINT;
	p_NtParamPPDec : UDINT;
	p_NtParamPPAutoSpd : UDINT;
	p_NtParamPPTuning : UDINT;
	p_NtParamPPMotorType : UDINT;
	p_NtParamProjCurtainSenPrep : UDINT;
	p_NtParamProjMagHeightChkPrep : UDINT;
	p_NtParamTravGotoMagWidthChkPt1 : UDINT;
	p_NtParamTravGotoMagWidthChkPt2 : UDINT;
	p_NtParamTravGotoMagWidthChkPt3 : UDINT;
	p_NtParamPPTorqParam : UDINT;
	p_NtParamProjLifTravMnlLoad : UDINT;
	p_NtParamCustomerReq : UDINT;
	p_NtParamProjShutter2Prep : UDINT;
	p_NtParamProjShutter3Prep : UDINT;
	p_NtParamAutoRcpPrep : UDINT;
	p_NtParamAutoRcpParamLmt : UDINT;
	p_NtParamAutoRcpPrecededBy : UDINT;
	p_NtParmProjChinesePrep : UDINT;
	p_NtParmProjGermanPrep : UDINT;
	p_NtParamProjOutShutter2Prep : UDINT;
	p_NtParamProjCntrPullLmt : UDINT;
	p_NtParamTrolleyLckPrep : UDINT;
	p_NtParamTrolleyLckProgNm : UDINT;
	p_NtParamTrolleyLckTwoCtrlIn : UDINT;
	p_NtParamTrolleyLckExtTO : UDINT;
	p_NtParamTrolleyLckRetTO : UDINT;
	p_NtParamTrolleyLckProgNm2 : UDINT;
	p_NtParamTrolleyLckTwoCtrlIn2 : UDINT;
	p_NtParamTrolleyLckExtTO2 : UDINT;
	p_NtParamTrolleyLckRetTO2 : UDINT;
END_VAR
(**)
(**)
```

### Program Logical/NtParam/NtParam

#### Act_Alarm.st
```iecst
(** 2019-03-25 **)
ACTION Act_Alarm:

	//Error
	IF EDGEPOS(eStatus = Error) THEN

		tyAlmData.sProgNm		:= p_sProgNm;
		tyAlmData.udiCode		:= udiStatus;
		tyAlmData.eSeverity		:= AlmSeverityError;
		tyAlmData.udiRunTime	:= tyAlmData.udiRunTime + 1;
		tyAlmData.bAlm			:= TRUE;
		tyAlmData.udiModuleNum  := udiModuleNum;
		g_sNtParamProgNm		:= p_sProgNm;
		//Get Error Message
		IF tyAlmData.udiCode < 10000 OR tyAlmData.udiCode > 10099 THEN
			tyAlmData.sAlmMsg	:= 'Unknown';
			tyAlmData.sRcyMsg	:= 'Unknown';
		ELSE
			tyAlmData.sAlmMsg	:= a_tyAlmText[tyAlmData.udiCode].sAlmText;
			tyAlmData.sRcyMsg	:= a_tyAlmText[tyAlmData.udiCode].sRcyText;
		END_IF

		sStatTxt	:= tyAlmData.sAlmMsg;

	ELSIF bRstErr AND (tyAlmData.udiCode <> 0) THEN

		tyAlmData.udiCode	:= 0;
		tyAlmData.eSeverity	:= AlmSeverityNA;
		tyAlmData.sAlmMsg	:= '';
		tyAlmData.sRcyMsg	:= '';
		tyAlmData.bAlm			:= FALSE;
		sStatTxt	:= a_sStatText[eStat];

	END_IF

END_ACTION
```

#### Act_InitGlobal.st
```iecst
(** 2019-03-25 **)
ACTION Act_InitGlobal:

	(* Always Change If Project Change *)

	//Pass Data To Link
	p_bLinkStartupRun ACCESS p_StartupRun;
	//Pass Data To Internal Use
	p_udiRstErr ACCESS p_RstErrReset;
	p_bSimu ACCESS p_UISimuMod;

	(* Always Change If Project Change *)

END_ACTION
```
